//     Enc/Inputs/In/nDataIn1[0] <-> ENC Status compact/Counter value
//     Enc/Inputs/In/nDataIn2[0] <-> ENC Status compact/Latch value
//     Enc/Inputs/In/nState1 @bit 4 <-> ENC Status compact/Status/Counter overflow
//     Enc/Inputs/In/nState1 @bit 3 <-> ENC Status compact/Status/Counter underflow
//     Enc/Inputs/In/nState1 @bit 7 <-> ENC Status compact/Status/Extrapolation stall
//     Enc/Inputs/In/nState1 <-> ENC Status compact/Status/Latch C valid
//     Enc/Inputs/In/nState1 @bit 1 <-> ENC Status compact/Status/Latch extern valid
//     Enc/Inputs/In/nState1 @bit 2 <-> ENC Status compact/Status/Set counter done
//     Enc/Inputs/In/nState2 @bit 4 <-> ENC Status compact/Status/Status of extern latch
//     Enc/Inputs/In/nState2 <-> ENC Status compact/Status/Status of input A
//     Enc/Inputs/In/nState2 @bit 1 <-> ENC Status compact/Status/Status of input B
//     Enc/Inputs/In/nState2 @bit 2 <-> ENC Status compact/Status/Status of input C
//     Enc/Inputs/In/nState2 @bit 5 <-> ENC Status compact/Status/Sync error
//     Enc/Inputs/In/nState2 @bit 7 <-> ENC Status compact/Status/TxPDO Toggle
//     Enc/Inputs/In/nState4 @bit 1 <-> WcState/InputToggle
//     Enc/Inputs/In/nState4 <-> WcState/WcState
//     Enc/Outputs/Out/nCtrl1 <-> ENC Control compact/Control/Enable latch C
//     Enc/Outputs/Out/nCtrl1 @bit 3 <-> ENC Control compact/Control/Enable latch extern on negative edge
//     Enc/Outputs/Out/nCtrl1 @bit 1 <-> ENC Control compact/Control/Enable latch extern on positive edge
//     Enc/Outputs/Out/nCtrl1 @bit 2 <-> ENC Control compact/Control/Set counter
//     Enc/Outputs/Out/nDataOut1[0] <-> ENC Control compact/Set counter value
//   (this object) <-> Device 1 (EtherCAT)/Term 5 (EK1200)/Term 6 (EK1122-0080)/DRL02-EK0 (EK1101-0080)/DRL02-E21 (EL7041)
//     Drive/Inputs/In/nState1 @bit 3 <-> STM Status/Status/Error
//     Drive/Inputs/In/nState1 @bit 5 <-> STM Status/Status/Moving negative
//     Drive/Inputs/In/nState1 @bit 4 <-> STM Status/Status/Moving positive
//     Drive/Inputs/In/nState1 @bit 1 <-> STM Status/Status/Ready
//     Drive/Inputs/In/nState1 <-> STM Status/Status/Ready to enable
//     Drive/Inputs/In/nState1 @bit 6 <-> STM Status/Status/Torque reduced
//     Drive/Inputs/In/nState1 @bit 2 <-> STM Status/Status/Warning
//     Drive/Inputs/In/nState2 @bit 3 <-> STM Status/Status/Digital input 1
//     Drive/Inputs/In/nState2 @bit 4 <-> STM Status/Status/Digital input 2
//     Drive/Inputs/In/nState2 @bit 5 <-> STM Status/Status/Sync error
//     Drive/Inputs/In/nState2 @bit 7 <-> STM Status/Status/TxPDO Toggle
//     Drive/Inputs/In/nState4 @bit 1 <-> WcState/InputToggle
//     Drive/Inputs/In/nState4 <-> WcState/WcState
//     Drive/Outputs/Out/nCtrl1 <-> STM Control/Control/Enable
//     Drive/Outputs/Out/nCtrl1 @bit 2 <-> STM Control/Control/Reduce torque
//     Drive/Outputs/Out/nCtrl1 @bit 1 <-> STM Control/Control/Reset
//     Drive/Outputs/Out/nDataOut2[0] <-> STM Velocity/Velocity
//     Enc/Inputs/In/nDataIn1[0] <-> ENC Status compact/Counter value
//     Enc/Inputs/In/nDataIn2[0] <-> ENC Status compact/Latch value
//     Enc/Inputs/In/nState1 @bit 4 <-> ENC Status compact/Status/Counter overflow
//     Enc/Inputs/In/nState1 @bit 3 <-> ENC Status compact/Status/Counter underflow
//     Enc/Inputs/In/nState1 @bit 7 <-> ENC Status compact/Status/Extrapolation stall
//     Enc/Inputs/In/nState1 <-> ENC Status compact/Status/Latch C valid
//     Enc/Inputs/In/nState1 @bit 1 <-> ENC Status compact/Status/Latch extern valid
//     Enc/Inputs/In/nState1 @bit 2 <-> ENC Status compact/Status/Set counter done
//     Enc/Inputs/In/nState2 @bit 4 <-> ENC Status compact/Status/Status of extern latch
//     Enc/Inputs/In/nState2 <-> ENC Status compact/Status/Status of input A
//     Enc/Inputs/In/nState2 @bit 1 <-> ENC Status compact/Status/Status of input B
//     Enc/Inputs/In/nState2 @bit 2 <-> ENC Status compact/Status/Status of input C
//     Enc/Inputs/In/nState2 @bit 5 <-> ENC Status compact/Status/Sync error
//     Enc/Inputs/In/nState2 @bit 7 <-> ENC Status compact/Status/TxPDO Toggle
//     Enc/Inputs/In/nState4 @bit 1 <-> WcState/InputToggle
//     Enc/Inputs/In/nState4 <-> WcState/WcState
//     Enc/Outputs/Out/nCtrl1 <-> ENC Control compact/Control/Enable latch C
//     Enc/Outputs/Out/nCtrl1 @bit 3 <-> ENC Control compact/Control/Enable latch extern on negative edge
//     Enc/Outputs/Out/nCtrl1 @bit 1 <-> ENC Control compact/Control/Enable latch extern on positive edge
//     Enc/Outputs/Out/nCtrl1 @bit 2 <-> ENC Control compact/Control/Set counter
//     Enc/Outputs/Out/nDataOut1[0] <-> ENC Control compact/Set counter value
//   (this object) <-> Device 1 (EtherCAT)/Term 5 (EK1200)/Term 6 (EK1122-0080)/DRL02-EK0 (EK1101-0080)/DRL02-E1 (EL7031)
//     Drive/Inputs/In/nState1 @bit 3 <-> STM Status/Status/Error
//     Drive/Inputs/In/nState1 @bit 5 <-> STM Status/Status/Moving negative
//     Drive/Inputs/In/nState1 @bit 4 <-> STM Status/Status/Moving positive
//     Drive/Inputs/In/nState1 @bit 1 <-> STM Status/Status/Ready
//     Drive/Inputs/In/nState1 <-> STM Status/Status/Ready to enable
//     Drive/Inputs/In/nState1 @bit 6 <-> STM Status/Status/Torque reduced
//     Drive/Inputs/In/nState1 @bit 2 <-> STM Status/Status/Warning
//     Drive/Inputs/In/nState2 @bit 3 <-> STM Status/Status/Digital input 1
//     Drive/Inputs/In/nState2 @bit 4 <-> STM Status/Status/Digital input 2
//     Drive/Inputs/In/nState2 @bit 5 <-> STM Status/Status/Sync error
//     Drive/Inputs/In/nState2 @bit 7 <-> STM Status/Status/TxPDO Toggle
//     Drive/Inputs/In/nState4 @bit 1 <-> WcState/InputToggle
//     Drive/Inputs/In/nState4 <-> WcState/WcState
//     Drive/Outputs/Out/nCtrl1 <-> STM Control/Control/Enable
//     Drive/Outputs/Out/nCtrl1 @bit 2 <-> STM Control/Control/Reduce torque
//     Drive/Outputs/Out/nCtrl1 @bit 1 <-> STM Control/Control/Reset
//     Drive/Outputs/Out/nDataOut2[0] <-> STM Velocity/Velocity
//   (this object) <-> Device 1 (EtherCAT)/Term 5 (EK1200)/Term 6 (EK1122-0080)/DRL02-EK0 (EK1101-0080)/DRL02-E2 (EL5042)
//     Enc/Inputs/In/nComState @bit 1 <-> WcState/InputToggle
//     Enc/Inputs/In/nComState <-> WcState/WcState
//     Enc/Inputs/In/nDataIn1 <-> FB Inputs Channel 1/Position
//     Enc/Inputs/In/nDataIn1 <-> FB Inputs Channel 2/Position
//     Enc/Inputs/In/nState1 @bit 12 <-> FB Inputs Channel 1/Status/Diag
//     Enc/Inputs/In/nState1 @bit 12 <-> FB Inputs Channel 2/Status/Diag
//     Enc/Inputs/In/nState1 @bit 1 <-> FB Inputs Channel 1/Status/Error
//     Enc/Inputs/In/nState1 @bit 1 <-> FB Inputs Channel 2/Status/Error
//     Enc/Inputs/In/nState1 @bit 14 <-> FB Inputs Channel 1/Status/Input cycle counter
//     Enc/Inputs/In/nState1 @bit 14 <-> FB Inputs Channel 2/Status/Input cycle counter
//     Enc/Inputs/In/nState1 @bit 2 <-> FB Inputs Channel 1/Status/Ready
//     Enc/Inputs/In/nState1 @bit 2 <-> FB Inputs Channel 2/Status/Ready
//     Enc/Inputs/In/nState1 @bit 13 <-> FB Inputs Channel 1/Status/TxPDO State
//     Enc/Inputs/In/nState1 @bit 13 <-> FB Inputs Channel 2/Status/TxPDO State
//     Enc/Inputs/In/nState1 <-> FB Inputs Channel 1/Status/Warning
//     Enc/Inputs/In/nState1 <-> FB Inputs Channel 2/Status/Warning
//   (this object) <-> Device 1 (EtherCAT)/Term 5 (EK1200)/Term 6 (EK1122-0080)/DRL02-EK0 (EK1101-0080)/DRL02-E3 (EL7031)
//     Drive/Inputs/In/nState1 @bit 3 <-> STM Status/Status/Error
//     Drive/Inputs/In/nState1 @bit 5 <-> STM Status/Status/Moving negative
//     Drive/Inputs/In/nState1 @bit 4 <-> STM Status/Status/Moving positive
//     Drive/Inputs/In/nState1 @bit 1 <-> STM Status/Status/Ready
//     Drive/Inputs/In/nState1 <-> STM Status/Status/Ready to enable
//     Drive/Inputs/In/nState1 @bit 6 <-> STM Status/Status/Torque reduced
//     Drive/Inputs/In/nState1 @bit 2 <-> STM Status/Status/Warning
//     Drive/Inputs/In/nState2 @bit 3 <-> STM Status/Status/Digital input 1
//     Drive/Inputs/In/nState2 @bit 4 <-> STM Status/Status/Digital input 2
//     Drive/Inputs/In/nState2 @bit 5 <-> STM Status/Status/Sync error
//     Drive/Inputs/In/nState2 @bit 7 <-> STM Status/Status/TxPDO Toggle
//     Drive/Inputs/In/nState4 @bit 1 <-> WcState/InputToggle
//     Drive/Inputs/In/nState4 <-> WcState/WcState
//     Drive/Outputs/Out/nCtrl1 <-> STM Control/Control/Enable
//     Drive/Outputs/Out/nCtrl1 @bit 2 <-> STM Control/Control/Reduce torque
//     Drive/Outputs/Out/nCtrl1 @bit 1 <-> STM Control/Control/Reset
//     Drive/Outputs/Out/nDataOut2[0] <-> STM Velocity/Velocity
//   (this object) <-> Device 1 (EtherCAT)/Term 5 (EK1200)/Term 6 (EK1122-0080)/DRL02-EK0 (EK1101-0080)/DRL02-E4 (EL7031)
//     Drive/Inputs/In/nState1 @bit 3 <-> STM Status/Status/Error
//     Drive/Inputs/In/nState1 @bit 5 <-> STM Status/Status/Moving negative
//     Drive/Inputs/In/nState1 @bit 4 <-> STM Status/Status/Moving positive
//     Drive/Inputs/In/nState1 @bit 1 <-> STM Status/Status/Ready
//     Drive/Inputs/In/nState1 <-> STM Status/Status/Ready to enable
//     Drive/Inputs/In/nState1 @bit 6 <-> STM Status/Status/Torque reduced
//     Drive/Inputs/In/nState1 @bit 2 <-> STM Status/Status/Warning
//     Drive/Inputs/In/nState2 @bit 3 <-> STM Status/Status/Digital input 1
//     Drive/Inputs/In/nState2 @bit 4 <-> STM Status/Status/Digital input 2
//     Drive/Inputs/In/nState2 @bit 5 <-> STM Status/Status/Sync error
//     Drive/Inputs/In/nState2 @bit 7 <-> STM Status/Status/TxPDO Toggle
//     Drive/Inputs/In/nState4 @bit 1 <-> WcState/InputToggle
//     Drive/Inputs/In/nState4 <-> WcState/WcState
//     Drive/Outputs/Out/nCtrl1 <-> STM Control/Control/Enable
//     Drive/Outputs/Out/nCtrl1 @bit 2 <-> STM Control/Control/Reduce torque
//     Drive/Outputs/Out/nCtrl1 @bit 1 <-> STM Control/Control/Reset
//     Drive/Outputs/Out/nDataOut2[0] <-> STM Velocity/Velocity
//   (this object) <-> Device 1 (EtherCAT)/Term 5 (EK1200)/Term 6 (EK1122-0080)/DRL02-EK0 (EK1101-0080)/DRL02-E5 (EL5042)
//     Enc/Inputs/In/nComState @bit 1 <-> WcState/InputToggle
//     Enc/Inputs/In/nComState <-> WcState/WcState
//     Enc/Inputs/In/nDataIn1 <-> FB Inputs Channel 1/Position
//     Enc/Inputs/In/nDataIn1 <-> FB Inputs Channel 2/Position
//     Enc/Inputs/In/nState1 @bit 12 <-> FB Inputs Channel 1/Status/Diag
//     Enc/Inputs/In/nState1 @bit 12 <-> FB Inputs Channel 2/Status/Diag
//     Enc/Inputs/In/nState1 @bit 1 <-> FB Inputs Channel 1/Status/Error
//     Enc/Inputs/In/nState1 @bit 1 <-> FB Inputs Channel 2/Status/Error
//     Enc/Inputs/In/nState1 @bit 14 <-> FB Inputs Channel 1/Status/Input cycle counter
//     Enc/Inputs/In/nState1 @bit 14 <-> FB Inputs Channel 2/Status/Input cycle counter
//     Enc/Inputs/In/nState1 @bit 2 <-> FB Inputs Channel 1/Status/Ready
//     Enc/Inputs/In/nState1 @bit 2 <-> FB Inputs Channel 2/Status/Ready
//     Enc/Inputs/In/nState1 @bit 13 <-> FB Inputs Channel 1/Status/TxPDO State
//     Enc/Inputs/In/nState1 @bit 13 <-> FB Inputs Channel 2/Status/TxPDO State
//     Enc/Inputs/In/nState1 <-> FB Inputs Channel 1/Status/Warning
//     Enc/Inputs/In/nState1 <-> FB Inputs Channel 2/Status/Warning
//   (this object) <-> Device 1 (EtherCAT)/Term 5 (EK1200)/Term 6 (EK1122-0080)/DRL02-EK0 (EK1101-0080)/DRL02-E6 (EL7031)
//     Drive/Inputs/In/nState1 @bit 3 <-> STM Status/Status/Error
//     Drive/Inputs/In/nState1 @bit 5 <-> STM Status/Status/Moving negative
//     Drive/Inputs/In/nState1 @bit 4 <-> STM Status/Status/Moving positive
//     Drive/Inputs/In/nState1 @bit 1 <-> STM Status/Status/Ready
//     Drive/Inputs/In/nState1 <-> STM Status/Status/Ready to enable
//     Drive/Inputs/In/nState1 @bit 6 <-> STM Status/Status/Torque reduced
//     Drive/Inputs/In/nState1 @bit 2 <-> STM Status/Status/Warning
//     Drive/Inputs/In/nState2 @bit 3 <-> STM Status/Status/Digital input 1
//     Drive/Inputs/In/nState2 @bit 4 <-> STM Status/Status/Digital input 2
//     Drive/Inputs/In/nState2 @bit 5 <-> STM Status/Status/Sync error
//     Drive/Inputs/In/nState2 @bit 7 <-> STM Status/Status/TxPDO Toggle
//     Drive/Inputs/In/nState4 @bit 1 <-> WcState/InputToggle
//     Drive/Inputs/In/nState4 <-> WcState/WcState
//     Drive/Outputs/Out/nCtrl1 <-> STM Control/Control/Enable
//     Drive/Outputs/Out/nCtrl1 @bit 2 <-> STM Control/Control/Reduce torque
//     Drive/Outputs/Out/nCtrl1 @bit 1 <-> STM Control/Control/Reset
//     Drive/Outputs/Out/nDataOut2[0] <-> STM Velocity/Velocity
//   (this object) <-> Device 1 (EtherCAT)/Term 5 (EK1200)/Term 6 (EK1122-0080)/DRL02-EK0 (EK1101-0080)/DRL02-E7 (EL7031)
//     Drive/Inputs/In/nState1 @bit 3 <-> STM Status/Status/Error
//     Drive/Inputs/In/nState1 @bit 5 <-> STM Status/Status/Moving negative
//     Drive/Inputs/In/nState1 @bit 4 <-> STM Status/Status/Moving positive
//     Drive/Inputs/In/nState1 @bit 1 <-> STM Status/Status/Ready
//     Drive/Inputs/In/nState1 <-> STM Status/Status/Ready to enable
//     Drive/Inputs/In/nState1 @bit 6 <-> STM Status/Status/Torque reduced
//     Drive/Inputs/In/nState1 @bit 2 <-> STM Status/Status/Warning
//     Drive/Inputs/In/nState2 @bit 3 <-> STM Status/Status/Digital input 1
//     Drive/Inputs/In/nState2 @bit 4 <-> STM Status/Status/Digital input 2
//     Drive/Inputs/In/nState2 @bit 5 <-> STM Status/Status/Sync error
//     Drive/Inputs/In/nState2 @bit 7 <-> STM Status/Status/TxPDO Toggle
//     Drive/Inputs/In/nState4 @bit 1 <-> WcState/InputToggle
//     Drive/Inputs/In/nState4 <-> WcState/WcState
//     Drive/Outputs/Out/nCtrl1 <-> STM Control/Control/Enable
//     Drive/Outputs/Out/nCtrl1 @bit 2 <-> STM Control/Control/Reduce torque
//     Drive/Outputs/Out/nCtrl1 @bit 1 <-> STM Control/Control/Reset
//     Drive/Outputs/Out/nDataOut2[0] <-> STM Velocity/Velocity
//   (this object) <-> Device 1 (EtherCAT)/Term 5 (EK1200)/Term 6 (EK1122-0080)/DRL02-EK0 (EK1101-0080)/DRL02-E8 (EL5042)
//     Enc/Inputs/In/nComState @bit 1 <-> WcState/InputToggle
//     Enc/Inputs/In/nComState <-> WcState/WcState
//     Enc/Inputs/In/nDataIn1 <-> FB Inputs Channel 1/Position
//     Enc/Inputs/In/nDataIn1 <-> FB Inputs Channel 2/Position
//     Enc/Inputs/In/nState1 @bit 12 <-> FB Inputs Channel 1/Status/Diag
//     Enc/Inputs/In/nState1 @bit 12 <-> FB Inputs Channel 2/Status/Diag
//     Enc/Inputs/In/nState1 @bit 1 <-> FB Inputs Channel 1/Status/Error
//     Enc/Inputs/In/nState1 @bit 1 <-> FB Inputs Channel 2/Status/Error
//     Enc/Inputs/In/nState1 @bit 14 <-> FB Inputs Channel 1/Status/Input cycle counter
//     Enc/Inputs/In/nState1 @bit 14 <-> FB Inputs Channel 2/Status/Input cycle counter
//     Enc/Inputs/In/nState1 @bit 2 <-> FB Inputs Channel 1/Status/Ready
//     Enc/Inputs/In/nState1 @bit 2 <-> FB Inputs Channel 2/Status/Ready
//     Enc/Inputs/In/nState1 @bit 13 <-> FB Inputs Channel 1/Status/TxPDO State
//     Enc/Inputs/In/nState1 @bit 13 <-> FB Inputs Channel 2/Status/TxPDO State
//     Enc/Inputs/In/nState1 <-> FB Inputs Channel 1/Status/Warning
//     Enc/Inputs/In/nState1 <-> FB Inputs Channel 2/Status/Warning
//   (this object) <-> Device 1 (EtherCAT)/Term 5 (EK1200)/Term 6 (EK1122-0080)/DRL02-EK0 (EK1101-0080)/DRL02-E9 (EL7031)
//     Drive/Inputs/In/nState1 @bit 3 <-> STM Status/Status/Error
//     Drive/Inputs/In/nState1 @bit 5 <-> STM Status/Status/Moving negative
//     Drive/Inputs/In/nState1 @bit 4 <-> STM Status/Status/Moving positive
//     Drive/Inputs/In/nState1 @bit 1 <-> STM Status/Status/Ready
//     Drive/Inputs/In/nState1 <-> STM Status/Status/Ready to enable
//     Drive/Inputs/In/nState1 @bit 6 <-> STM Status/Status/Torque reduced
//     Drive/Inputs/In/nState1 @bit 2 <-> STM Status/Status/Warning
//     Drive/Inputs/In/nState2 @bit 3 <-> STM Status/Status/Digital input 1
//     Drive/Inputs/In/nState2 @bit 4 <-> STM Status/Status/Digital input 2
//     Drive/Inputs/In/nState2 @bit 5 <-> STM Status/Status/Sync error
//     Drive/Inputs/In/nState2 @bit 7 <-> STM Status/Status/TxPDO Toggle
//     Drive/Inputs/In/nState4 @bit 1 <-> WcState/InputToggle
//     Drive/Inputs/In/nState4 <-> WcState/WcState
//     Drive/Outputs/Out/nCtrl1 <-> STM Control/Control/Enable
//     Drive/Outputs/Out/nCtrl1 @bit 2 <-> STM Control/Control/Reduce torque
//     Drive/Outputs/Out/nCtrl1 @bit 1 <-> STM Control/Control/Reset
//     Drive/Outputs/Out/nDataOut2[0] <-> STM Velocity/Velocity
//   (this object) <-> Device 1 (EtherCAT)/Term 5 (EK1200)/Term 6 (EK1122-0080)/DRL02-EK0 (EK1101-0080)/DRL02-E11 (EL7031)
//     Drive/Inputs/In/nState1 @bit 3 <-> STM Status/Status/Error
//     Drive/Inputs/In/nState1 @bit 5 <-> STM Status/Status/Moving negative
//     Drive/Inputs/In/nState1 @bit 4 <-> STM Status/Status/Moving positive
//     Drive/Inputs/In/nState1 @bit 1 <-> STM Status/Status/Ready
//     Drive/Inputs/In/nState1 <-> STM Status/Status/Ready to enable
//     Drive/Inputs/In/nState1 @bit 6 <-> STM Status/Status/Torque reduced
//     Drive/Inputs/In/nState1 @bit 2 <-> STM Status/Status/Warning
//     Drive/Inputs/In/nState2 @bit 3 <-> STM Status/Status/Digital input 1
//     Drive/Inputs/In/nState2 @bit 4 <-> STM Status/Status/Digital input 2
//     Drive/Inputs/In/nState2 @bit 5 <-> STM Status/Status/Sync error
//     Drive/Inputs/In/nState2 @bit 7 <-> STM Status/Status/TxPDO Toggle
//     Drive/Inputs/In/nState4 @bit 1 <-> WcState/InputToggle
//     Drive/Inputs/In/nState4 <-> WcState/WcState
//     Drive/Outputs/Out/nCtrl1 <-> STM Control/Control/Enable
//     Drive/Outputs/Out/nCtrl1 @bit 2 <-> STM Control/Control/Reduce torque
//     Drive/Outputs/Out/nCtrl1 @bit 1 <-> STM Control/Control/Reset
//     Drive/Outputs/Out/nDataOut2[0] <-> STM Velocity/Velocity
//   (this object) <-> Device 1 (EtherCAT)/Term 5 (EK1200)/Term 6 (EK1122-0080)/DRL02-EK0 (EK1101-0080)/DRL02-E12 (EL5042)
//     Enc/Inputs/In/nComState @bit 1 <-> WcState/InputToggle
//     Enc/Inputs/In/nComState <-> WcState/WcState
//     Enc/Inputs/In/nDataIn1 <-> FB Inputs Channel 1/Position
//     Enc/Inputs/In/nDataIn1 <-> FB Inputs Channel 2/Position
//     Enc/Inputs/In/nState1 @bit 12 <-> FB Inputs Channel 1/Status/Diag
//     Enc/Inputs/In/nState1 @bit 12 <-> FB Inputs Channel 2/Status/Diag
//     Enc/Inputs/In/nState1 @bit 1 <-> FB Inputs Channel 1/Status/Error
//     Enc/Inputs/In/nState1 @bit 1 <-> FB Inputs Channel 2/Status/Error
//     Enc/Inputs/In/nState1 @bit 14 <-> FB Inputs Channel 1/Status/Input cycle counter
//     Enc/Inputs/In/nState1 @bit 14 <-> FB Inputs Channel 2/Status/Input cycle counter
//     Enc/Inputs/In/nState1 @bit 2 <-> FB Inputs Channel 1/Status/Ready
//     Enc/Inputs/In/nState1 @bit 2 <-> FB Inputs Channel 2/Status/Ready
//     Enc/Inputs/In/nState1 @bit 13 <-> FB Inputs Channel 1/Status/TxPDO State
//     Enc/Inputs/In/nState1 @bit 13 <-> FB Inputs Channel 2/Status/TxPDO State
//     Enc/Inputs/In/nState1 <-> FB Inputs Channel 1/Status/Warning
//     Enc/Inputs/In/nState1 <-> FB Inputs Channel 2/Status/Warning
//   (this object) <-> Device 1 (EtherCAT)/Term 5 (EK1200)/Term 6 (EK1122-0080)/DRL02-EK0 (EK1101-0080)/DRL02-E13 (EL7041)
//     Drive/Inputs/In/nState1 @bit 3 <-> STM Status/Status/Error
//     Drive/Inputs/In/nState1 @bit 5 <-> STM Status/Status/Moving negative
//     Drive/Inputs/In/nState1 @bit 4 <-> STM Status/Status/Moving positive
//     Drive/Inputs/In/nState1 @bit 1 <-> STM Status/Status/Ready
//     Drive/Inputs/In/nState1 <-> STM Status/Status/Ready to enable
//     Drive/Inputs/In/nState1 @bit 6 <-> STM Status/Status/Torque reduced
//     Drive/Inputs/In/nState1 @bit 2 <-> STM Status/Status/Warning
//     Drive/Inputs/In/nState2 @bit 3 <-> STM Status/Status/Digital input 1
//     Drive/Inputs/In/nState2 @bit 4 <-> STM Status/Status/Digital input 2
//     Drive/Inputs/In/nState2 @bit 5 <-> STM Status/Status/Sync error
//     Drive/Inputs/In/nState2 @bit 7 <-> STM Status/Status/TxPDO Toggle
//     Drive/Inputs/In/nState4 @bit 1 <-> WcState/InputToggle
//     Drive/Inputs/In/nState4 <-> WcState/WcState
//     Drive/Outputs/Out/nCtrl1 <-> STM Control/Control/Enable
//     Drive/Outputs/Out/nCtrl1 @bit 2 <-> STM Control/Control/Reduce torque
//     Drive/Outputs/Out/nCtrl1 @bit 1 <-> STM Control/Control/Reset
//     Drive/Outputs/Out/nDataOut2[0] <-> STM Velocity/Velocity
//   (this object) <-> Device 1 (EtherCAT)/Term 5 (EK1200)/Term 6 (EK1122-0080)/DRL02-EK0 (EK1101-0080)/Term 63 (EL7031)
//     Drive/Inputs/In/nState1 @bit 3 <-> STM Status/Status/Error
//     Drive/Inputs/In/nState1 @bit 5 <-> STM Status/Status/Moving negative
//     Drive/Inputs/In/nState1 @bit 4 <-> STM Status/Status/Moving positive
//     Drive/Inputs/In/nState1 @bit 1 <-> STM Status/Status/Ready
//     Drive/Inputs/In/nState1 <-> STM Status/Status/Ready to enable
//     Drive/Inputs/In/nState1 @bit 6 <-> STM Status/Status/Torque reduced
//     Drive/Inputs/In/nState1 @bit 2 <-> STM Status/Status/Warning
//     Drive/Inputs/In/nState2 @bit 3 <-> STM Status/Status/Digital input 1
//     Drive/Inputs/In/nState2 @bit 4 <-> STM Status/Status/Digital input 2
//     Drive/Inputs/In/nState2 @bit 5 <-> STM Status/Status/Sync error
//     Drive/Inputs/In/nState2 @bit 7 <-> STM Status/Status/TxPDO Toggle
//     Drive/Inputs/In/nState4 @bit 1 <-> WcState/InputToggle
//     Drive/Inputs/In/nState4 <-> WcState/WcState
//     Drive/Outputs/Out/nCtrl1 <-> STM Control/Control/Enable
//     Drive/Outputs/Out/nCtrl1 @bit 2 <-> STM Control/Control/Reduce torque
//     Drive/Outputs/Out/nCtrl1 @bit 1 <-> STM Control/Control/Reset
//     Drive/Outputs/Out/nDataOut2[0] <-> STM Velocity/Velocity
//     Enc/Inputs/In/nDataIn1[0] <-> ENC Status compact/Counter value
//     Enc/Inputs/In/nDataIn2[0] <-> ENC Status compact/Latch value
//     Enc/Inputs/In/nState1 @bit 4 <-> ENC Status compact/Status/Counter overflow
//     Enc/Inputs/In/nState1 @bit 3 <-> ENC Status compact/Status/Counter underflow
//     Enc/Inputs/In/nState1 @bit 1 <-> ENC Status compact/Status/Latch extern valid
//     Enc/Inputs/In/nState1 @bit 2 <-> ENC Status compact/Status/Set counter done
//     Enc/Inputs/In/nState2 @bit 4 <-> ENC Status compact/Status/Status of extern latch
//     Enc/Inputs/In/nState2 @bit 5 <-> ENC Status compact/Status/Sync error
//     Enc/Inputs/In/nState2 @bit 7 <-> ENC Status compact/Status/TxPDO Toggle
//     Enc/Inputs/In/nState4 @bit 1 <-> WcState/InputToggle
//     Enc/Inputs/In/nState4 <-> WcState/WcState
//     Enc/Outputs/Out/nCtrl1 @bit 3 <-> ENC Control compact/Control/Enable latch extern on negative edge
//     Enc/Outputs/Out/nCtrl1 @bit 1 <-> ENC Control compact/Control/Enable latch extern on positive edge
//     Enc/Outputs/Out/nCtrl1 @bit 2 <-> ENC Control compact/Control/Set counter
//     Enc/Outputs/Out/nDataOut1[0] <-> ENC Control compact/Set counter value
//   (this object) <-> Device 1 (EtherCAT)/Term 5 (EK1200)/Term 6 (EK1122-0080)/DRL02-EK0 (EK1101-0080)/Term 66 (EL7031)
//     Drive/Inputs/In/nState1 @bit 3 <-> STM Status/Status/Error
//     Drive/Inputs/In/nState1 @bit 5 <-> STM Status/Status/Moving negative
//     Drive/Inputs/In/nState1 @bit 4 <-> STM Status/Status/Moving positive
//     Drive/Inputs/In/nState1 @bit 1 <-> STM Status/Status/Ready
//     Drive/Inputs/In/nState1 <-> STM Status/Status/Ready to enable
//     Drive/Inputs/In/nState1 @bit 6 <-> STM Status/Status/Torque reduced
//     Drive/Inputs/In/nState1 @bit 2 <-> STM Status/Status/Warning
//     Drive/Inputs/In/nState2 @bit 3 <-> STM Status/Status/Digital input 1
//     Drive/Inputs/In/nState2 @bit 4 <-> STM Status/Status/Digital input 2
//     Drive/Inputs/In/nState2 @bit 5 <-> STM Status/Status/Sync error
//     Drive/Inputs/In/nState2 @bit 7 <-> STM Status/Status/TxPDO Toggle
//     Drive/Inputs/In/nState4 @bit 1 <-> WcState/InputToggle
//     Drive/Inputs/In/nState4 <-> WcState/WcState
//     Drive/Outputs/Out/nCtrl1 <-> STM Control/Control/Enable
//     Drive/Outputs/Out/nCtrl1 @bit 2 <-> STM Control/Control/Reduce torque
//     Drive/Outputs/Out/nCtrl1 @bit 1 <-> STM Control/Control/Reset
//     Drive/Outputs/Out/nDataOut2[0] <-> STM Velocity/Velocity
//     Enc/Inputs/In/nDataIn1[0] <-> ENC Status compact/Counter value
//     Enc/Inputs/In/nDataIn2[0] <-> ENC Status compact/Latch value
//     Enc/Inputs/In/nState1 @bit 4 <-> ENC Status compact/Status/Counter overflow
//     Enc/Inputs/In/nState1 @bit 3 <-> ENC Status compact/Status/Counter underflow
//     Enc/Inputs/In/nState1 @bit 1 <-> ENC Status compact/Status/Latch extern valid
//     Enc/Inputs/In/nState1 @bit 2 <-> ENC Status compact/Status/Set counter done
//     Enc/Inputs/In/nState2 @bit 4 <-> ENC Status compact/Status/Status of extern latch
//     Enc/Inputs/In/nState2 @bit 5 <-> ENC Status compact/Status/Sync error
//     Enc/Inputs/In/nState2 @bit 7 <-> ENC Status compact/Status/TxPDO Toggle
//     Enc/Inputs/In/nState4 @bit 1 <-> WcState/InputToggle
//     Enc/Inputs/In/nState4 <-> WcState/WcState
//     Enc/Outputs/Out/nCtrl1 @bit 3 <-> ENC Control compact/Control/Enable latch extern on negative edge
//     Enc/Outputs/Out/nCtrl1 @bit 1 <-> ENC Control compact/Control/Enable latch extern on positive edge
//     Enc/Outputs/Out/nCtrl1 @bit 2 <-> ENC Control compact/Control/Set counter
//     Enc/Outputs/Out/nDataOut1[0] <-> ENC Control compact/Set counter value
//   (this object) <-> Device 1 (EtherCAT)/Term 5 (EK1200)/Term 6 (EK1122-0080)/DRL02-EK0 (EK1101-0080)/Term 67 (EL7031)
//     Drive/Inputs/In/nState1 @bit 3 <-> STM Status/Status/Error
//     Drive/Inputs/In/nState1 @bit 5 <-> STM Status/Status/Moving negative
//     Drive/Inputs/In/nState1 @bit 4 <-> STM Status/Status/Moving positive
//     Drive/Inputs/In/nState1 @bit 1 <-> STM Status/Status/Ready
//     Drive/Inputs/In/nState1 <-> STM Status/Status/Ready to enable
//     Drive/Inputs/In/nState1 @bit 6 <-> STM Status/Status/Torque reduced
//     Drive/Inputs/In/nState1 @bit 2 <-> STM Status/Status/Warning
//     Drive/Inputs/In/nState2 @bit 3 <-> STM Status/Status/Digital input 1
//     Drive/Inputs/In/nState2 @bit 4 <-> STM Status/Status/Digital input 2
//     Drive/Inputs/In/nState2 @bit 5 <-> STM Status/Status/Sync error
//     Drive/Inputs/In/nState2 @bit 7 <-> STM Status/Status/TxPDO Toggle
//     Drive/Inputs/In/nState4 @bit 1 <-> WcState/InputToggle
//     Drive/Inputs/In/nState4 <-> WcState/WcState
//     Drive/Outputs/Out/nCtrl1 <-> STM Control/Control/Enable
//     Drive/Outputs/Out/nCtrl1 @bit 2 <-> STM Control/Control/Reduce torque
//     Drive/Outputs/Out/nCtrl1 @bit 1 <-> STM Control/Control/Reset
//     Drive/Outputs/Out/nDataOut2[0] <-> STM Velocity/Velocity
//     Enc/Inputs/In/nDataIn1[0] <-> ENC Status compact/Counter value
//     Enc/Inputs/In/nDataIn2[0] <-> ENC Status compact/Latch value
//     Enc/Inputs/In/nState1 @bit 4 <-> ENC Status compact/Status/Counter overflow
//     Enc/Inputs/In/nState1 @bit 3 <-> ENC Status compact/Status/Counter underflow
//     Enc/Inputs/In/nState1 @bit 1 <-> ENC Status compact/Status/Latch extern valid
//     Enc/Inputs/In/nState1 @bit 2 <-> ENC Status compact/Status/Set counter done
//     Enc/Inputs/In/nState2 @bit 4 <-> ENC Status compact/Status/Status of extern latch
//     Enc/Inputs/In/nState2 @bit 5 <-> ENC Status compact/Status/Sync error
//     Enc/Inputs/In/nState2 @bit 7 <-> ENC Status compact/Status/TxPDO Toggle
//     Enc/Inputs/In/nState4 @bit 1 <-> WcState/InputToggle
//     Enc/Inputs/In/nState4 <-> WcState/WcState
//     Enc/Outputs/Out/nCtrl1 @bit 3 <-> ENC Control compact/Control/Enable latch extern on negative edge
//     Enc/Outputs/Out/nCtrl1 @bit 1 <-> ENC Control compact/Control/Enable latch extern on positive edge
//     Enc/Outputs/Out/nCtrl1 @bit 2 <-> ENC Control compact/Control/Set counter
//     Enc/Outputs/Out/nDataOut1[0] <-> ENC Control compact/Set counter value
//   (this object) <-> Device 1 (EtherCAT)/Term 5 (EK1200)/Term 6 (EK1122-0080)/DRL02-EK0 (EK1101-0080)/DRL02-E17 (EL7031)
//     Drive/Inputs/In/nState1 @bit 3 <-> STM Status/Status/Error
//     Drive/Inputs/In/nState1 @bit 5 <-> STM Status/Status/Moving negative
//     Drive/Inputs/In/nState1 @bit 4 <-> STM Status/Status/Moving positive
//     Drive/Inputs/In/nState1 @bit 1 <-> STM Status/Status/Ready
//     Drive/Inputs/In/nState1 <-> STM Status/Status/Ready to enable
//     Drive/Inputs/In/nState1 @bit 6 <-> STM Status/Status/Torque reduced
//     Drive/Inputs/In/nState1 @bit 2 <-> STM Status/Status/Warning
//     Drive/Inputs/In/nState2 @bit 3 <-> STM Status/Status/Digital input 1
//     Drive/Inputs/In/nState2 @bit 4 <-> STM Status/Status/Digital input 2
//     Drive/Inputs/In/nState2 @bit 5 <-> STM Status/Status/Sync error
//     Drive/Inputs/In/nState2 @bit 7 <-> STM Status/Status/TxPDO Toggle
//     Drive/Inputs/In/nState4 @bit 1 <-> WcState/InputToggle
//     Drive/Inputs/In/nState4 <-> WcState/WcState
//     Drive/Outputs/Out/nCtrl1 <-> STM Control/Control/Enable
//     Drive/Outputs/Out/nCtrl1 @bit 2 <-> STM Control/Control/Reduce torque
//     Drive/Outputs/Out/nCtrl1 @bit 1 <-> STM Control/Control/Reset
//     Drive/Outputs/Out/nDataOut2[0] <-> STM Velocity/Velocity
//   (this object) <-> Device 1 (EtherCAT)/Term 5 (EK1200)/Term 6 (EK1122-0080)/DRL02-EK0 (EK1101-0080)/DRL02-E18 (EL5042)
//     Enc/Inputs/In/nComState @bit 1 <-> WcState/InputToggle
//     Enc/Inputs/In/nComState <-> WcState/WcState
//     Enc/Inputs/In/nDataIn1 <-> FB Inputs Channel 1/Position
//     Enc/Inputs/In/nDataIn1 <-> FB Inputs Channel 2/Position
//     Enc/Inputs/In/nState1 @bit 12 <-> FB Inputs Channel 1/Status/Diag
//     Enc/Inputs/In/nState1 @bit 12 <-> FB Inputs Channel 2/Status/Diag
//     Enc/Inputs/In/nState1 @bit 1 <-> FB Inputs Channel 1/Status/Error
//     Enc/Inputs/In/nState1 @bit 1 <-> FB Inputs Channel 2/Status/Error
//     Enc/Inputs/In/nState1 @bit 14 <-> FB Inputs Channel 1/Status/Input cycle counter
//     Enc/Inputs/In/nState1 @bit 14 <-> FB Inputs Channel 2/Status/Input cycle counter
//     Enc/Inputs/In/nState1 @bit 2 <-> FB Inputs Channel 1/Status/Ready
//     Enc/Inputs/In/nState1 @bit 2 <-> FB Inputs Channel 2/Status/Ready
//     Enc/Inputs/In/nState1 @bit 13 <-> FB Inputs Channel 1/Status/TxPDO State
//     Enc/Inputs/In/nState1 @bit 13 <-> FB Inputs Channel 2/Status/TxPDO State
//     Enc/Inputs/In/nState1 <-> FB Inputs Channel 1/Status/Warning
//     Enc/Inputs/In/nState1 <-> FB Inputs Channel 2/Status/Warning
//   (this object) <-> Device 1 (EtherCAT)/Term 5 (EK1200)/Term 6 (EK1122-0080)/DRL02-EK0 (EK1101-0080)/DRL02-E19 (EL7031)
//     Drive/Inputs/In/nState1 @bit 3 <-> STM Status/Status/Error
//     Drive/Inputs/In/nState1 @bit 5 <-> STM Status/Status/Moving negative
//     Drive/Inputs/In/nState1 @bit 4 <-> STM Status/Status/Moving positive
//     Drive/Inputs/In/nState1 @bit 1 <-> STM Status/Status/Ready
//     Drive/Inputs/In/nState1 <-> STM Status/Status/Ready to enable
//     Drive/Inputs/In/nState1 @bit 6 <-> STM Status/Status/Torque reduced
//     Drive/Inputs/In/nState1 @bit 2 <-> STM Status/Status/Warning
//     Drive/Inputs/In/nState2 @bit 3 <-> STM Status/Status/Digital input 1
//     Drive/Inputs/In/nState2 @bit 4 <-> STM Status/Status/Digital input 2
//     Drive/Inputs/In/nState2 @bit 5 <-> STM Status/Status/Sync error
//     Drive/Inputs/In/nState2 @bit 7 <-> STM Status/Status/TxPDO Toggle
//     Drive/Inputs/In/nState4 @bit 1 <-> WcState/InputToggle
//     Drive/Inputs/In/nState4 <-> WcState/WcState
//     Drive/Outputs/Out/nCtrl1 <-> STM Control/Control/Enable
//     Drive/Outputs/Out/nCtrl1 @bit 2 <-> STM Control/Control/Reduce torque
//     Drive/Outputs/Out/nCtrl1 @bit 1 <-> STM Control/Control/Reset
//     Drive/Outputs/Out/nDataOut2[0] <-> STM Velocity/Velocity
//   (this object) <-> Device 1 (EtherCAT)/Term 5 (EK1200)/Term 6 (EK1122-0080)/DRL02-EK0 (EK1101-0080)/DRL02-E24 (EL7031)
//     Drive/Inputs/In/nState1 @bit 3 <-> STM Status/Status/Error
//     Drive/Inputs/In/nState1 @bit 5 <-> STM Status/Status/Moving negative
//     Drive/Inputs/In/nState1 @bit 4 <-> STM Status/Status/Moving positive
//     Drive/Inputs/In/nState1 @bit 1 <-> STM Status/Status/Ready
//     Drive/Inputs/In/nState1 <-> STM Status/Status/Ready to enable
//     Drive/Inputs/In/nState1 @bit 6 <-> STM Status/Status/Torque reduced
//     Drive/Inputs/In/nState1 @bit 2 <-> STM Status/Status/Warning
//     Drive/Inputs/In/nState2 @bit 3 <-> STM Status/Status/Digital input 1
//     Drive/Inputs/In/nState2 @bit 4 <-> STM Status/Status/Digital input 2
//     Drive/Inputs/In/nState2 @bit 5 <-> STM Status/Status/Sync error
//     Drive/Inputs/In/nState2 @bit 7 <-> STM Status/Status/TxPDO Toggle
//     Drive/Inputs/In/nState4 @bit 1 <-> WcState/InputToggle
//     Drive/Inputs/In/nState4 <-> WcState/WcState
//     Drive/Outputs/Out/nCtrl1 <-> STM Control/Control/Enable
//     Drive/Outputs/Out/nCtrl1 @bit 2 <-> STM Control/Control/Reduce torque
//     Drive/Outputs/Out/nCtrl1 @bit 1 <-> STM Control/Control/Reset
//     Drive/Outputs/Out/nDataOut2[0] <-> STM Velocity/Velocity
//   (this object) <-> Device 1 (EtherCAT)/Term 5 (EK1200)/Term 6 (EK1122-0080)/DRL02-EK0 (EK1101-0080)/Term 91 (EL5112)
//     Enc/Inputs/In/nDataIn1 <-> ENC Status Channel 1/Counter value
//     Enc/Inputs/In/nDataIn2 <-> ENC Status Channel 1/Latch value
//     Enc/Inputs/In/nState1 @bit 4 <-> ENC Status Channel 1/Status/Counter overflow
//     Enc/Inputs/In/nState1 @bit 3 <-> ENC Status Channel 1/Status/Counter underflow
//     Enc/Inputs/In/nState1 @bit 1 <-> ENC Status Channel 1/Status/Latch extern valid
//     Enc/Inputs/In/nState1 @bit 6 <-> ENC Status Channel 1/Status/Open circuit
//     Enc/Inputs/In/nState1 @bit 2 <-> ENC Status Channel 1/Status/Set counter done
//     Enc/Inputs/In/nState2 <-> ENC Status Channel 1/Status/Status of input A
//     Enc/Inputs/In/nState2 @bit 1 <-> ENC Status Channel 1/Status/Status of input B
//     Enc/Inputs/In/nState2 @bit 3 <-> ENC Status Channel 1/Status/Status of input gate
//     Enc/Inputs/In/nState4 @bit 1 <-> WcState/InputToggle
//     Enc/Inputs/In/nState4 <-> WcState/WcState
//     Enc/Outputs/Out/nCtrl1 @bit 3 <-> ENC Control Channel 1/Control/Enable latch extern on negative edge
//     Enc/Outputs/Out/nCtrl1 @bit 1 <-> ENC Control Channel 1/Control/Enable latch extern on positive edge
//     Enc/Outputs/Out/nCtrl1 @bit 2 <-> ENC Control Channel 1/Control/Set counter
//     Enc/Outputs/Out/nCtrl2 @bit 2 <-> ENC Control Channel 1/Control/Set counter on latch extern on negative edge
//     Enc/Outputs/Out/nCtrl2 @bit 1 <-> ENC Control Channel 1/Control/Set counter on latch extern on positive edge
//     Enc/Outputs/Out/nCtrl2 <-> ENC Control Channel 1/Control/Set software gate
//     Enc/Outputs/Out/nDataOut1 <-> ENC Control Channel 1/Set counter value
//   (this object) <-> Device 1 (EtherCAT)/Term 5 (EK1200)/Term 6 (EK1122-0080)/DRL02-EK0 (EK1101-0080)/DRL02-E25 (EL5042)
//     Enc/Inputs/In/nComState @bit 1 <-> WcState/InputToggle
//     Enc/Inputs/In/nComState <-> WcState/WcState
//     Enc/Inputs/In/nDataIn1 <-> FB Inputs Channel 2/Position
//     Enc/Inputs/In/nState1 @bit 12 <-> FB Inputs Channel 2/Status/Diag
//     Enc/Inputs/In/nState1 @bit 1 <-> FB Inputs Channel 2/Status/Error
//     Enc/Inputs/In/nState1 @bit 14 <-> FB Inputs Channel 2/Status/Input cycle counter
//     Enc/Inputs/In/nState1 @bit 2 <-> FB Inputs Channel 2/Status/Ready
//     Enc/Inputs/In/nState1 @bit 13 <-> FB Inputs Channel 2/Status/TxPDO State
//     Enc/Inputs/In/nState1 <-> FB Inputs Channel 2/Status/Warning
//   (this object) <-> Device 1 (EtherCAT)/Term 5 (EK1200)/Term 6 (EK1122-0080)/DRL02-EK0 (EK1101-0080)/DRL02-E26 (EL7031)
//     Drive/Inputs/In/nState1 @bit 3 <-> STM Status/Status/Error
//     Drive/Inputs/In/nState1 @bit 5 <-> STM Status/Status/Moving negative
//     Drive/Inputs/In/nState1 @bit 4 <-> STM Status/Status/Moving positive
//     Drive/Inputs/In/nState1 @bit 1 <-> STM Status/Status/Ready
//     Drive/Inputs/In/nState1 <-> STM Status/Status/Ready to enable
//     Drive/Inputs/In/nState1 @bit 6 <-> STM Status/Status/Torque reduced
//     Drive/Inputs/In/nState1 @bit 2 <-> STM Status/Status/Warning
//     Drive/Inputs/In/nState2 @bit 3 <-> STM Status/Status/Digital input 1
//     Drive/Inputs/In/nState2 @bit 4 <-> STM Status/Status/Digital input 2
//     Drive/Inputs/In/nState2 @bit 5 <-> STM Status/Status/Sync error
//     Drive/Inputs/In/nState2 @bit 7 <-> STM Status/Status/TxPDO Toggle
//     Drive/Inputs/In/nState4 @bit 1 <-> WcState/InputToggle
//     Drive/Inputs/In/nState4 <-> WcState/WcState
//     Drive/Outputs/Out/nCtrl1 <-> STM Control/Control/Enable
//     Drive/Outputs/Out/nCtrl1 @bit 2 <-> STM Control/Control/Reduce torque
//     Drive/Outputs/Out/nCtrl1 @bit 1 <-> STM Control/Control/Reset
//     Drive/Outputs/Out/nDataOut2[0] <-> STM Velocity/Velocity
//   (this object) <-> Device 1 (EtherCAT)/Term 5 (EK1200)/Term 6 (EK1122-0080)/DRL02-EK0 (EK1101-0080)/DRL02-E27 (EL7031)
//     Drive/Inputs/In/nState1 @bit 3 <-> STM Status/Status/Error
//     Drive/Inputs/In/nState1 @bit 5 <-> STM Status/Status/Moving negative
//     Drive/Inputs/In/nState1 @bit 4 <-> STM Status/Status/Moving positive
//     Drive/Inputs/In/nState1 @bit 1 <-> STM Status/Status/Ready
//     Drive/Inputs/In/nState1 <-> STM Status/Status/Ready to enable
//     Drive/Inputs/In/nState1 @bit 6 <-> STM Status/Status/Torque reduced
//     Drive/Inputs/In/nState1 @bit 2 <-> STM Status/Status/Warning
//     Drive/Inputs/In/nState2 @bit 3 <-> STM Status/Status/Digital input 1
//     Drive/Inputs/In/nState2 @bit 4 <-> STM Status/Status/Digital input 2
//     Drive/Inputs/In/nState2 @bit 5 <-> STM Status/Status/Sync error
//     Drive/Inputs/In/nState2 @bit 7 <-> STM Status/Status/TxPDO Toggle
//     Drive/Inputs/In/nState4 @bit 1 <-> WcState/InputToggle
//     Drive/Inputs/In/nState4 <-> WcState/WcState
//     Drive/Outputs/Out/nCtrl1 <-> STM Control/Control/Enable
//     Drive/Outputs/Out/nCtrl1 @bit 2 <-> STM Control/Control/Reduce torque
//     Drive/Outputs/Out/nCtrl1 @bit 1 <-> STM Control/Control/Reset
//     Drive/Outputs/Out/nDataOut2[0] <-> STM Velocity/Velocity
//     Enc/Inputs/In/nDataIn1[0] <-> ENC Status compact/Counter value
//     Enc/Inputs/In/nDataIn2[0] <-> ENC Status compact/Latch value
//     Enc/Inputs/In/nState1 @bit 4 <-> ENC Status compact/Status/Counter overflow
//     Enc/Inputs/In/nState1 @bit 3 <-> ENC Status compact/Status/Counter underflow
//     Enc/Inputs/In/nState1 @bit 1 <-> ENC Status compact/Status/Latch extern valid
//     Enc/Inputs/In/nState1 @bit 2 <-> ENC Status compact/Status/Set counter done
//     Enc/Inputs/In/nState2 @bit 4 <-> ENC Status compact/Status/Status of extern latch
//     Enc/Inputs/In/nState2 @bit 5 <-> ENC Status compact/Status/Sync error
//     Enc/Inputs/In/nState2 @bit 7 <-> ENC Status compact/Status/TxPDO Toggle
//     Enc/Inputs/In/nState4 @bit 1 <-> WcState/InputToggle
//     Enc/Inputs/In/nState4 <-> WcState/WcState
//     Enc/Outputs/Out/nCtrl1 @bit 3 <-> ENC Control compact/Control/Enable latch extern on negative edge
//     Enc/Outputs/Out/nCtrl1 @bit 1 <-> ENC Control compact/Control/Enable latch extern on positive edge
//     Enc/Outputs/Out/nCtrl1 @bit 2 <-> ENC Control compact/Control/Set counter
//     Enc/Outputs/Out/nDataOut1[0] <-> ENC Control compact/Set counter value
//   (this object) <-> Device 1 (EtherCAT)/Term 5 (EK1200)/Term 6 (EK1122-0080)/DRL02-EK0 (EK1101-0080)/DRL02-E29 (EL7031)
//     Drive/Inputs/In/nState1 @bit 3 <-> STM Status/Status/Error
//     Drive/Inputs/In/nState1 @bit 5 <-> STM Status/Status/Moving negative
//     Drive/Inputs/In/nState1 @bit 4 <-> STM Status/Status/Moving positive
//     Drive/Inputs/In/nState1 @bit 1 <-> STM Status/Status/Ready
//     Drive/Inputs/In/nState1 <-> STM Status/Status/Ready to enable
//     Drive/Inputs/In/nState1 @bit 6 <-> STM Status/Status/Torque reduced
//     Drive/Inputs/In/nState1 @bit 2 <-> STM Status/Status/Warning
//     Drive/Inputs/In/nState2 @bit 3 <-> STM Status/Status/Digital input 1
//     Drive/Inputs/In/nState2 @bit 4 <-> STM Status/Status/Digital input 2
//     Drive/Inputs/In/nState2 @bit 5 <-> STM Status/Status/Sync error
//     Drive/Inputs/In/nState2 @bit 7 <-> STM Status/Status/TxPDO Toggle
//     Drive/Inputs/In/nState4 @bit 1 <-> WcState/InputToggle
//     Drive/Inputs/In/nState4 <-> WcState/WcState
//     Drive/Outputs/Out/nCtrl1 <-> STM Control/Control/Enable
//     Drive/Outputs/Out/nCtrl1 @bit 2 <-> STM Control/Control/Reduce torque
//     Drive/Outputs/Out/nCtrl1 @bit 1 <-> STM Control/Control/Reset
//     Drive/Outputs/Out/nDataOut2[0] <-> STM Velocity/Velocity
//     Enc/Inputs/In/nDataIn1[0] <-> ENC Status compact/Counter value
//     Enc/Inputs/In/nDataIn2[0] <-> ENC Status compact/Latch value
//     Enc/Inputs/In/nState1 @bit 4 <-> ENC Status compact/Status/Counter overflow
//     Enc/Inputs/In/nState1 @bit 3 <-> ENC Status compact/Status/Counter underflow
//     Enc/Inputs/In/nState1 @bit 1 <-> ENC Status compact/Status/Latch extern valid
//     Enc/Inputs/In/nState1 @bit 2 <-> ENC Status compact/Status/Set counter done
//     Enc/Inputs/In/nState2 @bit 4 <-> ENC Status compact/Status/Status of extern latch
//     Enc/Inputs/In/nState2 @bit 5 <-> ENC Status compact/Status/Sync error
//     Enc/Inputs/In/nState2 @bit 7 <-> ENC Status compact/Status/TxPDO Toggle
//     Enc/Inputs/In/nState4 @bit 1 <-> WcState/InputToggle
//     Enc/Inputs/In/nState4 <-> WcState/WcState
//     Enc/Outputs/Out/nCtrl1 @bit 3 <-> ENC Control compact/Control/Enable latch extern on negative edge
//     Enc/Outputs/Out/nCtrl1 @bit 1 <-> ENC Control compact/Control/Enable latch extern on positive edge
//     Enc/Outputs/Out/nCtrl1 @bit 2 <-> ENC Control compact/Control/Set counter
//     Enc/Outputs/Out/nDataOut1[0] <-> ENC Control compact/Set counter value
//   (this object) <-> Device 1 (EtherCAT)/Term 5 (EK1200)/Term 6 (EK1122-0080)/DRL02-EK0 (EK1101-0080)/DRL02-E30 (EL7031)
//     Drive/Inputs/In/nState1 @bit 3 <-> STM Status/Status/Error
//     Drive/Inputs/In/nState1 @bit 5 <-> STM Status/Status/Moving negative
//     Drive/Inputs/In/nState1 @bit 4 <-> STM Status/Status/Moving positive
//     Drive/Inputs/In/nState1 @bit 1 <-> STM Status/Status/Ready
//     Drive/Inputs/In/nState1 <-> STM Status/Status/Ready to enable
//     Drive/Inputs/In/nState1 @bit 6 <-> STM Status/Status/Torque reduced
//     Drive/Inputs/In/nState1 @bit 2 <-> STM Status/Status/Warning
//     Drive/Inputs/In/nState2 @bit 3 <-> STM Status/Status/Digital input 1
//     Drive/Inputs/In/nState2 @bit 4 <-> STM Status/Status/Digital input 2
//     Drive/Inputs/In/nState2 @bit 5 <-> STM Status/Status/Sync error
//     Drive/Inputs/In/nState2 @bit 7 <-> STM Status/Status/TxPDO Toggle
//     Drive/Inputs/In/nState4 @bit 1 <-> WcState/InputToggle
//     Drive/Inputs/In/nState4 <-> WcState/WcState
//     Drive/Outputs/Out/nCtrl1 <-> STM Control/Control/Enable
//     Drive/Outputs/Out/nCtrl1 @bit 2 <-> STM Control/Control/Reduce torque
//     Drive/Outputs/Out/nCtrl1 @bit 1 <-> STM Control/Control/Reset
//     Drive/Outputs/Out/nDataOut2[0] <-> STM Velocity/Velocity
//     Enc/Inputs/In/nDataIn1[0] <-> ENC Status compact/Counter value
//     Enc/Inputs/In/nDataIn2[0] <-> ENC Status compact/Latch value
//     Enc/Inputs/In/nState1 @bit 4 <-> ENC Status compact/Status/Counter overflow
//     Enc/Inputs/In/nState1 @bit 3 <-> ENC Status compact/Status/Counter underflow
//     Enc/Inputs/In/nState1 @bit 1 <-> ENC Status compact/Status/Latch extern valid
//     Enc/Inputs/In/nState1 @bit 2 <-> ENC Status compact/Status/Set counter done
//     Enc/Inputs/In/nState2 @bit 4 <-> ENC Status compact/Status/Status of extern latch
//     Enc/Inputs/In/nState2 @bit 5 <-> ENC Status compact/Status/Sync error
//     Enc/Inputs/In/nState2 @bit 7 <-> ENC Status compact/Status/TxPDO Toggle
//     Enc/Inputs/In/nState4 @bit 1 <-> WcState/InputToggle
//     Enc/Inputs/In/nState4 <-> WcState/WcState
//     Enc/Outputs/Out/nCtrl1 @bit 3 <-> ENC Control compact/Control/Enable latch extern on negative edge
//     Enc/Outputs/Out/nCtrl1 @bit 1 <-> ENC Control compact/Control/Enable latch extern on positive edge
//     Enc/Outputs/Out/nCtrl1 @bit 2 <-> ENC Control compact/Control/Set counter
//     Enc/Outputs/Out/nDataOut1[0] <-> ENC Control compact/Set counter value
//   (this object) <-> Device 1 (EtherCAT)/Term 5 (EK1200)/Term 6 (EK1122-0080)/DRL02-EK0 (EK1101-0080)/DRL02-E33 (EL7031)
//     Drive/Inputs/In/nState1 @bit 3 <-> STM Status/Status/Error
//     Drive/Inputs/In/nState1 @bit 5 <-> STM Status/Status/Moving negative
//     Drive/Inputs/In/nState1 @bit 4 <-> STM Status/Status/Moving positive
//     Drive/Inputs/In/nState1 @bit 1 <-> STM Status/Status/Ready
//     Drive/Inputs/In/nState1 <-> STM Status/Status/Ready to enable
//     Drive/Inputs/In/nState1 @bit 6 <-> STM Status/Status/Torque reduced
//     Drive/Inputs/In/nState1 @bit 2 <-> STM Status/Status/Warning
//     Drive/Inputs/In/nState2 @bit 3 <-> STM Status/Status/Digital input 1
//     Drive/Inputs/In/nState2 @bit 4 <-> STM Status/Status/Digital input 2
//     Drive/Inputs/In/nState2 @bit 5 <-> STM Status/Status/Sync error
//     Drive/Inputs/In/nState2 @bit 7 <-> STM Status/Status/TxPDO Toggle
//     Drive/Inputs/In/nState4 @bit 1 <-> WcState/InputToggle
//     Drive/Inputs/In/nState4 <-> WcState/WcState
//     Drive/Outputs/Out/nCtrl1 <-> STM Control/Control/Enable
//     Drive/Outputs/Out/nCtrl1 @bit 2 <-> STM Control/Control/Reduce torque
//     Drive/Outputs/Out/nCtrl1 @bit 1 <-> STM Control/Control/Reset
//     Drive/Outputs/Out/nDataOut2[0] <-> STM Velocity/Velocity
//   (this object) <-> Device 1 (EtherCAT)/Term 5 (EK1200)/Term 6 (EK1122-0080)/DRL02-EK0 (EK1101-0080)/DRL02-E31 (EL7031)
//     Drive/Inputs/In/nState1 @bit 3 <-> STM Status/Status/Error
//     Drive/Inputs/In/nState1 @bit 5 <-> STM Status/Status/Moving negative
//     Drive/Inputs/In/nState1 @bit 4 <-> STM Status/Status/Moving positive
//     Drive/Inputs/In/nState1 @bit 1 <-> STM Status/Status/Ready
//     Drive/Inputs/In/nState1 <-> STM Status/Status/Ready to enable
//     Drive/Inputs/In/nState1 @bit 6 <-> STM Status/Status/Torque reduced
//     Drive/Inputs/In/nState1 @bit 2 <-> STM Status/Status/Warning
//     Drive/Inputs/In/nState2 @bit 3 <-> STM Status/Status/Digital input 1
//     Drive/Inputs/In/nState2 @bit 4 <-> STM Status/Status/Digital input 2
//     Drive/Inputs/In/nState2 @bit 5 <-> STM Status/Status/Sync error
//     Drive/Inputs/In/nState2 @bit 7 <-> STM Status/Status/TxPDO Toggle
//     Drive/Inputs/In/nState4 @bit 1 <-> WcState/InputToggle
//     Drive/Inputs/In/nState4 <-> WcState/WcState
//     Drive/Outputs/Out/nCtrl1 <-> STM Control/Control/Enable
//     Drive/Outputs/Out/nCtrl1 @bit 2 <-> STM Control/Control/Reduce torque
//     Drive/Outputs/Out/nCtrl1 @bit 1 <-> STM Control/Control/Reset
//     Drive/Outputs/Out/nDataOut2[0] <-> STM Velocity/Velocity
//   (this object) <-> Device 1 (EtherCAT)/Term 5 (EK1200)/Term 6 (EK1122-0080)/DRL02-EK0 (EK1101-0080)/DRL02-E32 (EL5042)
//     Enc/Inputs/In/nComState @bit 1 <-> WcState/InputToggle
//     Enc/Inputs/In/nComState <-> WcState/WcState
//     Enc/Inputs/In/nDataIn1 <-> FB Inputs Channel 1/Position
//     Enc/Inputs/In/nState1 @bit 12 <-> FB Inputs Channel 1/Status/Diag
//     Enc/Inputs/In/nState1 @bit 1 <-> FB Inputs Channel 1/Status/Error
//     Enc/Inputs/In/nState1 @bit 14 <-> FB Inputs Channel 1/Status/Input cycle counter
//     Enc/Inputs/In/nState1 @bit 2 <-> FB Inputs Channel 1/Status/Ready
//     Enc/Inputs/In/nState1 @bit 13 <-> FB Inputs Channel 1/Status/TxPDO State
//     Enc/Inputs/In/nState1 <-> FB Inputs Channel 1/Status/Warning
//   (this object) <-> Device 1 (EtherCAT)/Term 5 (EK1200)/Term 6 (EK1122-0080)/DRL02-EK0 (EK1101-0080)/DRL02-E28 (EL5042)
//     Enc/Inputs/In/nComState @bit 1 <-> WcState/InputToggle
//     Enc/Inputs/In/nComState <-> WcState/WcState
//     Enc/Inputs/In/nDataIn1 <-> FB Inputs Channel 1/Position
//     Enc/Inputs/In/nState1 @bit 12 <-> FB Inputs Channel 1/Status/Diag
//     Enc/Inputs/In/nState1 @bit 1 <-> FB Inputs Channel 1/Status/Error
//     Enc/Inputs/In/nState1 @bit 14 <-> FB Inputs Channel 1/Status/Input cycle counter
//     Enc/Inputs/In/nState1 @bit 2 <-> FB Inputs Channel 1/Status/Ready
//     Enc/Inputs/In/nState1 @bit 13 <-> FB Inputs Channel 1/Status/TxPDO State
//     Enc/Inputs/In/nState1 <-> FB Inputs Channel 1/Status/Warning
//   PLC_CRIX_MOT Instance <-> Device 1 (EtherCAT)/Term 5 (EK1200)/Term 167 (EK1122)/CRIX_VAC_INTF (EL6695-0002)
//     PlcTask Inputs/PRG_CryoPump.bCRYO_VGC_01_CLS <-> IO Inputs/bCRYO_VGC_01_CLS
//     PlcTask Inputs/PRG_CryoPump.bCRYO_VGC_02_CLS <-> IO Inputs/bCRYO_VGC_02_CLS
//     PlcTask Inputs/PRG_CryoPump.bCRYO_VGC_01_OPN <-> IO Inputs/bCRYO_VGC_01_OPN
//     PlcTask Inputs/PRG_CryoPump.bCRYO_VGC_02_OPN <-> IO Inputs/bCRYO_VGC_02_OPN
//     PlcTask Inputs/PRG_CryoPump.xEcatBridge_TxPDO_state <-> SYNC Inputs/TxPDO state
//     PlcTask Inputs/PRG_CryoPump.xEcatBridge_WcState <-> WcState/WcState
//     PlcTask Inputs/PRG_InjectorMotors.bSDS_VGC_01_CLS <-> IO Inputs/bSDS_VGC_01_CLS
//     PlcTask Inputs/PRG_InjectorMotors.bSDS_VGC_01_OPN <-> IO Inputs/bSDS_VGC_01_OPN
//     PlcTask Outputs/PRG_CryoPump.bMOTY10_IN <-> IO Outputs/bMOTY10_IN
//     PlcTask Outputs/PRG_CryoPump.bMOTY11_IN <-> IO Outputs/bMOTY11_IN
//     PlcTask Outputs/PRG_CryoPump.bMOTY10_OUT <-> IO Outputs/bMOTY10_OUT
//     PlcTask Outputs/PRG_CryoPump.bMOTY11_OUT <-> IO Outputs/bMOTY11_OUT
//     PlcTask Outputs/PRG_InjectorMotors.bMOTSDSZ18_IN <-> IO Outputs/bMOTSDSZ18_IN
//     PlcTask Outputs/PRG_InjectorMotors.bMOTSDSZ18_OUT <-> IO Outputs/bMOTSDSZ18_OUT
//   PLC_CRIX_MOT Instance <-> Device 1 (EtherCAT)/Term 5 (EK1200)/Term 6 (EK1122-0080)/DRL02-EK0 (EK1101-0080)/DRL02-E1 (EL7031)
//     PlcTask Inputs/Main.M1.bLimitBackwardEnable <-> STM Status/Status/Digital input 1
//     PlcTask Inputs/Main.M1.bLimitForwardEnable <-> STM Status/Status/Digital input 2
//   PLC_CRIX_MOT Instance <-> Device 1 (EtherCAT)/Term 5 (EK1200)/Term 6 (EK1122-0080)/DRL02-EK0 (EK1101-0080)/DRL02-E11 (EL7031)
//     PlcTask Inputs/Main.M7.bLimitBackwardEnable <-> STM Status/Status/Digital input 2
//     PlcTask Inputs/Main.M7.bLimitForwardEnable <-> STM Status/Status/Digital input 1
//   PLC_CRIX_MOT Instance <-> Device 1 (EtherCAT)/Term 5 (EK1200)/Term 6 (EK1122-0080)/DRL02-EK0 (EK1101-0080)/DRL02-E13 (EL7041)
//     PlcTask Inputs/Main.M8.bLimitBackwardEnable <-> STM Status/Status/Digital input 2
//     PlcTask Inputs/Main.M8.bLimitForwardEnable <-> STM Status/Status/Digital input 1
//   PLC_CRIX_MOT Instance <-> Device 1 (EtherCAT)/Term 5 (EK1200)/Term 6 (EK1122-0080)/DRL02-EK0 (EK1101-0080)/DRL02-E17 (EL7031)
//     PlcTask Inputs/Main.M12.bLimitBackwardEnable <-> STM Status/Status/Digital input 2
//     PlcTask Inputs/Main.M12.bLimitForwardEnable <-> STM Status/Status/Digital input 1
//   PLC_CRIX_MOT Instance <-> Device 1 (EtherCAT)/Term 5 (EK1200)/Term 6 (EK1122-0080)/DRL02-EK0 (EK1101-0080)/DRL02-E19 (EL7031)
//     PlcTask Inputs/Main.M13.bLimitBackwardEnable <-> STM Status/Status/Digital input 2
//     PlcTask Inputs/Main.M13.bLimitForwardEnable <-> STM Status/Status/Digital input 1
//   PLC_CRIX_MOT Instance <-> Device 1 (EtherCAT)/Term 5 (EK1200)/Term 6 (EK1122-0080)/DRL02-EK0 (EK1101-0080)/DRL02-E21 (EL7041)
//     PlcTask Inputs/Main.M49.bLimitForwardEnable <-> STM Status/Status/Digital input 2
//     PlcTask Inputs/PRG_CryoPump.bLimitBackwardEnable_Y_11 <-> STM Status/Status/Digital input 1
//   PLC_CRIX_MOT Instance <-> Device 1 (EtherCAT)/Term 5 (EK1200)/Term 6 (EK1122-0080)/DRL02-EK0 (EK1101-0080)/DRL02-E23 (EL7041)
//     PlcTask Inputs/Main.M48.bLimitForwardEnable <-> STM Status/Status/Digital input 2
//     PlcTask Inputs/PRG_CryoPump.bLimitBackwardEnable_Y_10 <-> STM Status/Status/Digital input 1
//   PLC_CRIX_MOT Instance <-> Device 1 (EtherCAT)/Term 5 (EK1200)/Term 6 (EK1122-0080)/DRL02-EK0 (EK1101-0080)/DRL02-E26 (EL7031)
//     PlcTask Inputs/Main.M17.bLimitBackwardEnable <-> STM Status/Status/Digital input 2
//     PlcTask Inputs/Main.M17.bLimitForwardEnable <-> STM Status/Status/Digital input 1
//   PLC_CRIX_MOT Instance <-> Device 1 (EtherCAT)/Term 5 (EK1200)/Term 6 (EK1122-0080)/DRL02-EK0 (EK1101-0080)/DRL02-E27 (EL7031)
//     PlcTask Inputs/Main.M18.bLimitForwardEnable <-> STM Status/Status/Digital input 1
//     PlcTask Inputs/PRG_InjectorMotors.bLimitBackwardEnable_SDSZ_18 <-> STM Status/Status/Digital input 2
//   PLC_CRIX_MOT Instance <-> Device 1 (EtherCAT)/Term 5 (EK1200)/Term 6 (EK1122-0080)/DRL02-EK0 (EK1101-0080)/DRL02-E3 (EL7031)
//     PlcTask Inputs/Main.M2.bLimitBackwardEnable <-> STM Status/Status/Digital input 2
//     PlcTask Inputs/Main.M2.bLimitForwardEnable <-> STM Status/Status/Digital input 1
//   PLC_CRIX_MOT Instance <-> Device 1 (EtherCAT)/Term 5 (EK1200)/Term 6 (EK1122-0080)/DRL02-EK0 (EK1101-0080)/DRL02-E31 (EL7031)
//     PlcTask Inputs/Main.M35.bLimitBackwardEnable <-> STM Status/Status/Digital input 2
//     PlcTask Inputs/Main.M35.bLimitForwardEnable <-> STM Status/Status/Digital input 1
//   PLC_CRIX_MOT Instance <-> Device 1 (EtherCAT)/Term 5 (EK1200)/Term 6 (EK1122-0080)/DRL02-EK0 (EK1101-0080)/DRL02-E4 (EL7031)
//     PlcTask Inputs/Main.M3.bLimitBackwardEnable <-> STM Status/Status/Digital input 2
//     PlcTask Inputs/Main.M3.bLimitForwardEnable <-> STM Status/Status/Digital input 1
//   PLC_CRIX_MOT Instance <-> Device 1 (EtherCAT)/Term 5 (EK1200)/Term 6 (EK1122-0080)/DRL02-EK0 (EK1101-0080)/DRL02-E6 (EL7031)
//     PlcTask Inputs/Main.M4.bLimitBackwardEnable <-> STM Status/Status/Digital input 1
//     PlcTask Inputs/Main.M4.bLimitForwardEnable <-> STM Status/Status/Digital input 2
//   PLC_CRIX_MOT Instance <-> Device 1 (EtherCAT)/Term 5 (EK1200)/Term 6 (EK1122-0080)/DRL02-EK0 (EK1101-0080)/DRL02-E7 (EL7031)
//     PlcTask Inputs/Main.M5.bLimitBackwardEnable <-> STM Status/Status/Digital input 2
//     PlcTask Inputs/Main.M5.bLimitForwardEnable <-> STM Status/Status/Digital input 1
//   PLC_CRIX_MOT Instance <-> Device 1 (EtherCAT)/Term 5 (EK1200)/Term 6 (EK1122-0080)/DRL02-EK0 (EK1101-0080)/DRL02-E9 (EL7031)
//     PlcTask Inputs/Main.M6.bLimitBackwardEnable <-> STM Status/Status/Digital input 2
//     PlcTask Inputs/Main.M6.bLimitForwardEnable <-> STM Status/Status/Digital input 1
//   PLC_CRIX_MOT Instance <-> Device 1 (EtherCAT)/Term 5 (EK1200)/Term 6 (EK1122-0080)/DRL02-EK0 (EK1101-0080)/DRL02-ECJ0 (EK1122-0080)/Term 109 (EK1101-0080)/Camera X (EL7041)
//     PlcTask Inputs/Main.M33.bLimitBackwardEnable <-> STM Status/Status/Digital input 2
//     PlcTask Inputs/Main.M33.bLimitForwardEnable <-> STM Status/Status/Digital input 1
//   PLC_CRIX_MOT Instance <-> Device 1 (EtherCAT)/Term 5 (EK1200)/Term 6 (EK1122-0080)/DRL02-EK0 (EK1101-0080)/DRL02-ECJ0 (EK1122-0080)/Term 109 (EK1101-0080)/Camera Y (EL7041)
//     PlcTask Inputs/Main.M34.bLimitBackwardEnable <-> STM Status/Status/Digital input 2
//     PlcTask Inputs/Main.M34.bLimitForwardEnable <-> STM Status/Status/Digital input 1
//   PLC_CRIX_MOT Instance <-> Device 1 (EtherCAT)/Term 5 (EK1200)/Term 6 (EK1122-0080)/DRL02-EK0 (EK1101-0080)/DRL02-ECJ0 (EK1122-0080)/Term 113 (EK1101-0080)/Beamblock X (EL7041)
//     PlcTask Inputs/Main.M30.bLimitBackwardEnable <-> STM Status/Status/Digital input 2
//     PlcTask Inputs/Main.M30.bLimitForwardEnable <-> STM Status/Status/Digital input 1
//   PLC_CRIX_MOT Instance <-> Device 1 (EtherCAT)/Term 5 (EK1200)/Term 6 (EK1122-0080)/DRL02-EK0 (EK1101-0080)/DRL02-ECJ0 (EK1122-0080)/Term 113 (EK1101-0080)/Beamblock Y (EL7041)
//     PlcTask Inputs/Main.M31.bLimitBackwardEnable <-> STM Status/Status/Digital input 2
//     PlcTask Inputs/Main.M31.bLimitForwardEnable <-> STM Status/Status/Digital input 1
//   PLC_CRIX_MOT Instance <-> Device 1 (EtherCAT)/Term 5 (EK1200)/Term 6 (EK1122-0080)/DRL02-EK0 (EK1101-0080)/DRL02-ECJ0 (EK1122-0080)/Term 113 (EK1101-0080)/Beamblock Z (EL7041)
//     PlcTask Inputs/Main.M32.bLimitBackwardEnable <-> STM Status/Status/Digital input 2
//     PlcTask Inputs/Main.M32.bLimitForwardEnable <-> STM Status/Status/Digital input 1
//   PLC_CRIX_MOT Instance <-> Device 1 (EtherCAT)/Term 5 (EK1200)/Term 6 (EK1122-0080)/DRL02-EK0 (EK1101-0080)/DRL02-ECJ1 (EK1122)/CryoStat (EK1101)/Cryo X (EL7041)
//     PlcTask Inputs/Main.M22.bLimitBackwardEnable <-> STM Status/Status/Digital input 2
//     PlcTask Inputs/Main.M22.bLimitForwardEnable <-> STM Status/Status/Digital input 1
//   PLC_CRIX_MOT Instance <-> Device 1 (EtherCAT)/Term 5 (EK1200)/Term 6 (EK1122-0080)/DRL02-EK0 (EK1101-0080)/DRL02-ECJ1 (EK1122)/CryoStat (EK1101)/Cryo Y (EL7041)
//     PlcTask Inputs/Main.M23.bLimitBackwardEnable <-> STM Status/Status/Digital input 2
//     PlcTask Inputs/Main.M23.bLimitForwardEnable <-> STM Status/Status/Digital input 1
//   PLC_CRIX_MOT Instance <-> Device 1 (EtherCAT)/Term 5 (EK1200)/Term 6 (EK1122-0080)/DRL02-EK0 (EK1101-0080)/DRL02-ECJ1 (EK1122)/CryoStat (EK1101)/Cryo Z (EL7041)
//     PlcTask Inputs/Main.M24.bLimitBackwardEnable <-> STM Status/Status/Digital input 2
//     PlcTask Inputs/Main.M24.bLimitForwardEnable <-> STM Status/Status/Digital input 1
//   PLC_CRIX_MOT Instance <-> Device 1 (EtherCAT)/Term 5 (EK1200)/Term 6 (EK1122-0080)/DRL02-EK0 (EK1101-0080)/DRL02-ECJ1 (EK1122)/CryoStat (EK1101)/Term 158 (EL4004)
//     PlcTask Outputs/GVL_FiberLite.bLedOutput1.iIlluminatorINT <-> AO Outputs Channel 1/Analog output
//   PLC_CRIX_MOT Instance <-> Device 1 (EtherCAT)/Term 5 (EK1200)/Term 6 (EK1122-0080)/DRL02-EK0 (EK1101-0080)/DRL02-ECJ1 (EK1122)/VLS_EP10_EP7041-3102
//     PlcTask Inputs/Main.M44.bHome <-> ENC Status compact/Status/Status of input C
//     PlcTask Inputs/Main.M44.bLimitBackwardEnable <-> STM Status/Status/Digital input 1
//     PlcTask Inputs/Main.M44.bLimitForwardEnable <-> STM Status/Status/Digital input 2
//     PlcTask Inputs/Main.M44.nRawEncoderUINT <-> ENC Status compact/Counter value
//   PLC_CRIX_MOT Instance <-> Device 1 (EtherCAT)/Term 5 (EK1200)/Term 6 (EK1122-0080)/DRL02-EK0 (EK1101-0080)/DRL02-ECJ1 (EK1122)/VLS_EP11_EP7041-3102
//     PlcTask Inputs/Main.M45.bHome <-> ENC Status compact/Status/Status of input C
//     PlcTask Inputs/Main.M45.bLimitBackwardEnable <-> STM Status/Status/Digital input 1
//     PlcTask Inputs/Main.M45.bLimitForwardEnable <-> STM Status/Status/Digital input 2
//     PlcTask Inputs/Main.M45.nRawEncoderUINT <-> ENC Status compact/Counter value
//   PLC_CRIX_MOT Instance <-> Device 1 (EtherCAT)/Term 5 (EK1200)/Term 6 (EK1122-0080)/DRL02-EK0 (EK1101-0080)/DRL02-ECJ1 (EK1122)/VLS_EP12_EP7041-3102
//     PlcTask Inputs/Main.M46.bHome <-> ENC Status compact/Status/Status of input C
//     PlcTask Inputs/Main.M46.bLimitBackwardEnable <-> STM Status/Status/Digital input 2
//     PlcTask Inputs/Main.M46.bLimitForwardEnable <-> STM Status/Status/Digital input 1
//   PLC_CRIX_MOT Instance <-> Device 1 (EtherCAT)/Term 5 (EK1200)/Term 6 (EK1122-0080)/DRL02-EK0 (EK1101-0080)/DRL02-ECJ1 (EK1122)/VLS_EP13_EP7041-3102
//     PlcTask Inputs/Main.M47.bHome <-> ENC Status compact/Status/Status of input C
//     PlcTask Inputs/Main.M47.bLimitBackwardEnable <-> STM Status/Status/Digital input 1
//     PlcTask Inputs/Main.M47.bLimitForwardEnable <-> STM Status/Status/Digital input 2
//   PLC_CRIX_MOT Instance <-> Device 1 (EtherCAT)/Term 5 (EK1200)/Term 6 (EK1122-0080)/DRL02-EK0 (EK1101-0080)/DRL02-ECJ1 (EK1122)/VLS_EP6_EP7041-1002
//     PlcTask Inputs/Main.M40.bLimitBackwardEnable <-> STM Status/Status/Digital input 2
//     PlcTask Inputs/Main.M40.bLimitForwardEnable <-> STM Status/Status/Digital input 1
//   PLC_CRIX_MOT Instance <-> Device 1 (EtherCAT)/Term 5 (EK1200)/Term 6 (EK1122-0080)/DRL02-EK0 (EK1101-0080)/DRL02-ECJ1 (EK1122)/VLS_EP7_EP7041-1002
//     PlcTask Inputs/Main.M41.bLimitBackwardEnable <-> STM Status/Status/Digital input 2
//     PlcTask Inputs/Main.M41.bLimitForwardEnable <-> STM Status/Status/Digital input 1
//   PLC_CRIX_MOT Instance <-> Device 1 (EtherCAT)/Term 5 (EK1200)/Term 6 (EK1122-0080)/DRL02-EK0 (EK1101-0080)/DRL02-ECJ1 (EK1122)/VLS_EP8_EP7041-1002
//     PlcTask Inputs/Main.M42.bLimitBackwardEnable <-> STM Status/Status/Digital input 2
//     PlcTask Inputs/Main.M42.bLimitForwardEnable <-> STM Status/Status/Digital input 1
//   PLC_CRIX_MOT Instance <-> Device 1 (EtherCAT)/Term 5 (EK1200)/Term 6 (EK1122-0080)/DRL02-EK0 (EK1101-0080)/DRL02-ECJ1 (EK1122)/VLS_EP9_EP7041-1002
//     PlcTask Inputs/Main.M43.bLimitBackwardEnable <-> STM Status/Status/Digital input 2
//     PlcTask Inputs/Main.M43.bLimitForwardEnable <-> STM Status/Status/Digital input 1
//   PLC_CRIX_MOT Instance <-> Device 1 (EtherCAT)/Term 5 (EK1200)/Term 6 (EK1122-0080)/DRL02-EK0 (EK1101-0080)/DRL02-ECJ2 (EK1122)/Catcher (EK1100)/Catcher_E1_EL7041
//     PlcTask Inputs/Main.M37.bLimitBackwardEnable <-> STM Status/Status/Digital input 1
//     PlcTask Inputs/Main.M37.bLimitForwardEnable <-> STM Status/Status/Digital input 2
//   PLC_CRIX_MOT Instance <-> Device 1 (EtherCAT)/Term 5 (EK1200)/Term 6 (EK1122-0080)/DRL02-EK0 (EK1101-0080)/DRL02-ECJ2 (EK1122)/Catcher (EK1100)/Catcher_E3_EL7041
//     PlcTask Inputs/Main.M38.bLimitBackwardEnable <-> STM Status/Status/Digital input 2
//     PlcTask Inputs/Main.M38.bLimitForwardEnable <-> STM Status/Status/Digital input 1
//   PLC_CRIX_MOT Instance <-> Device 1 (EtherCAT)/Term 5 (EK1200)/Term 6 (EK1122-0080)/DRL02-EK0 (EK1101-0080)/DRL02-ECJ2 (EK1122)/Catcher (EK1100)/Catcher_E4_EL7041
//     PlcTask Inputs/Main.M39.bLimitBackwardEnable <-> STM Status/Status/Digital input 1
//     PlcTask Inputs/Main.M39.bLimitForwardEnable <-> STM Status/Status/Digital input 2
//   PLC_CRIX_MOT Instance <-> Device 1 (EtherCAT)/Term 5 (EK1200)/Term 6 (EK1122-0080)/DRL02-EK0 (EK1101-0080)/Term 173 (EL1124)
//     PlcTask Inputs/PRG_InjectorMotors.bHall_Backward <-> Channel 4/Input
//     PlcTask Inputs/PRG_InjectorMotors.bHall_Forward <-> Channel 3/Input
//   PLC_CRIX_MOT Instance <-> Device 1 (EtherCAT)/Term 5 (EK1200)/Term 6 (EK1122-0080)/DRL02-EK0 (EK1101-0080)/Term 65 (EL1084)
//     PlcTask Inputs/Main.M10.bLimitBackwardEnable <-> Channel 4/Input
//     PlcTask Inputs/Main.M9.bLimitBackwardEnable <-> Channel 2/Input
//     PlcTask Inputs/Main.M10.bLimitForwardEnable <-> Channel 3/Input
//     PlcTask Inputs/Main.M9.bLimitForwardEnable <-> Channel 1/Input
//   PLC_CRIX_MOT Instance <-> Device 1 (EtherCAT)/Term 5 (EK1200)/Term 6 (EK1122-0080)/DRL02-EK0 (EK1101-0080)/Term 68 (EL1084)
//     PlcTask Inputs/Main.M11.bLimitBackwardEnable <-> Channel 2/Input
//     PlcTask Inputs/Main.M11.bLimitForwardEnable <-> Channel 1/Input
//   PLC_CRIX_MOT Instance <-> Device 1 (EtherCAT)/Term 5 (EK1200)/Term 83 (EK1521-0010)/Term 166 (EK1501-0010)/PMPS_FFO
//     PlcTask Outputs/GVL_PMPS.g_FastFaultOutput1.q_xFastFaultOut <-> Channel 1/Output
//     PlcTask Outputs/GVL_PMPS.g_FastFaultOutput2.q_xFastFaultOut <-> Channel 2/Output
//   PLC_CRIX_MOT Instance <-> Device 1 (EtherCAT)/Term 5 (EK1200)/Term 83 (EK1521-0010)/Term 166 (EK1501-0010)/PMPS_PRE
//     PlcTask Inputs/PRG_PMPS.fbArbiterIO.i_stCurrentBP <-> IO Inputs/CurrentBP
//     PlcTask Inputs/PRG_PMPS.fbArbiterIO.xTxPDO_state <-> SYNC Inputs/TxPDO state
//     PlcTask Inputs/PRG_PMPS.fbArbiterIO.xTxPDO_toggle <-> SYNC Inputs/TxPDO toggle
//     PlcTask Outputs/PRG_PMPS.fbArbiterIO.q_stRequestedBP <-> IO Outputs/RequestedBP
//   PLC_CRIX_MOT Instance <-> NC-Task 1 SAF/Axes/Axis 1 - Diagnostic Paddle X
//     PlcTask Inputs/Main.M1.Axis.NcToPlc <-> Outputs/ToPlc
//     PlcTask Outputs/Main.M1.Axis.PlcToNc <-> Inputs/FromPlc
//   PLC_CRIX_MOT Instance <-> NC-Task 1 SAF/Axes/Axis 10 - Illumination Y
//     PlcTask Inputs/Main.M10.Axis.NcToPlc <-> Outputs/ToPlc
//     PlcTask Outputs/Main.M10.Axis.PlcToNc <-> Inputs/FromPlc
//   PLC_CRIX_MOT Instance <-> NC-Task 1 SAF/Axes/Axis 11 - Illumination Z
//     PlcTask Inputs/Main.M11.Axis.NcToPlc <-> Outputs/ToPlc
//     PlcTask Outputs/Main.M11.Axis.PlcToNc <-> Inputs/FromPlc
//   PLC_CRIX_MOT Instance <-> NC-Task 1 SAF/Axes/Axis 12 - Questar X
//     PlcTask Inputs/Main.M12.Axis.NcToPlc <-> Outputs/ToPlc
//     PlcTask Outputs/Main.M12.Axis.PlcToNc <-> Inputs/FromPlc
//   PLC_CRIX_MOT Instance <-> NC-Task 1 SAF/Axes/Axis 13 - Questar Y
//     PlcTask Inputs/Main.M13.Axis.NcToPlc <-> Outputs/ToPlc
//     PlcTask Outputs/Main.M13.Axis.PlcToNc <-> Inputs/FromPlc
//   PLC_CRIX_MOT Instance <-> NC-Task 1 SAF/Axes/Axis 14 - SPARE 1
//     PlcTask Inputs/Main.M14.Axis.NcToPlc <-> Outputs/ToPlc
//     PlcTask Outputs/Main.M14.Axis.PlcToNc <-> Inputs/FromPlc
//   PLC_CRIX_MOT Instance <-> NC-Task 1 SAF/Axes/Axis 15 - SPARE 2
//     PlcTask Inputs/Main.M15.Axis.NcToPlc <-> Outputs/ToPlc
//     PlcTask Outputs/Main.M15.Axis.PlcToNc <-> Inputs/FromPlc
//   PLC_CRIX_MOT Instance <-> NC-Task 1 SAF/Axes/Axis 16 - SDS Injector X
//     PlcTask Inputs/Main.M16.Axis.NcToPlc <-> Outputs/ToPlc
//     PlcTask Outputs/Main.M16.Axis.PlcToNc <-> Inputs/FromPlc
//   PLC_CRIX_MOT Instance <-> NC-Task 1 SAF/Axes/Axis 17 - SDS Injectory Y
//     PlcTask Inputs/Main.M17.Axis.NcToPlc <-> Outputs/ToPlc
//     PlcTask Outputs/Main.M17.Axis.PlcToNc <-> Inputs/FromPlc
//   PLC_CRIX_MOT Instance <-> NC-Task 1 SAF/Axes/Axis 18 - SDS Injector Z
//     PlcTask Inputs/Main.M18.Axis.NcToPlc <-> Outputs/ToPlc
//     PlcTask Outputs/Main.M18.Axis.PlcToNc <-> Inputs/FromPlc
//   PLC_CRIX_MOT Instance <-> NC-Task 1 SAF/Axes/Axis 19 - SDS Rotation Y
//     PlcTask Inputs/Main.M19.Axis.NcToPlc <-> Outputs/ToPlc
//     PlcTask Outputs/Main.M19.Axis.PlcToNc <-> Inputs/FromPlc
//   PLC_CRIX_MOT Instance <-> NC-Task 1 SAF/Axes/Axis 2 - Diagnostic Paddle Y
//     PlcTask Inputs/Main.M2.Axis.NcToPlc <-> Outputs/ToPlc
//     PlcTask Outputs/Main.M2.Axis.PlcToNc <-> Inputs/FromPlc
//   PLC_CRIX_MOT Instance <-> NC-Task 1 SAF/Axes/Axis 20 - SDS Shroud Rotation
//     PlcTask Inputs/Main.M20.Axis.NcToPlc <-> Outputs/ToPlc
//     PlcTask Outputs/Main.M20.Axis.PlcToNc <-> Inputs/FromPlc
//   PLC_CRIX_MOT Instance <-> NC-Task 1 SAF/Axes/Axis 3 - Diagnostic Paddle Z
//     PlcTask Inputs/Main.M3.Axis.NcToPlc <-> Outputs/ToPlc
//     PlcTask Outputs/Main.M3.Axis.PlcToNc <-> Inputs/FromPlc
//   PLC_CRIX_MOT Instance <-> NC-Task 1 SAF/Axes/Axis 35 - Outcoupling Lens Y
//     PlcTask Inputs/Main.M35.Axis.NcToPlc <-> Outputs/ToPlc
//     PlcTask Outputs/Main.M35.Axis.PlcToNc <-> Inputs/FromPlc
//   PLC_CRIX_MOT Instance <-> NC-Task 1 SAF/Axes/Axis 36 - SDS Z Encoder
//     PlcTask Inputs/Main.M36.Axis.NcToPlc <-> Outputs/ToPlc
//     PlcTask Outputs/Main.M36.Axis.PlcToNc <-> Inputs/FromPlc
//   PLC_CRIX_MOT Instance <-> NC-Task 1 SAF/Axes/Axis 4 - Objectives X
//     PlcTask Inputs/Main.M4.Axis.NcToPlc <-> Outputs/ToPlc
//     PlcTask Outputs/Main.M4.Axis.PlcToNc <-> Inputs/FromPlc
//   PLC_CRIX_MOT Instance <-> NC-Task 1 SAF/Axes/Axis 5 - Objectives Y
//     PlcTask Inputs/Main.M5.Axis.NcToPlc <-> Outputs/ToPlc
//     PlcTask Outputs/Main.M5.Axis.PlcToNc <-> Inputs/FromPlc
//   PLC_CRIX_MOT Instance <-> NC-Task 1 SAF/Axes/Axis 6 - Objectives Z
//     PlcTask Inputs/Main.M6.Axis.NcToPlc <-> Outputs/ToPlc
//     PlcTask Outputs/Main.M6.Axis.PlcToNc <-> Inputs/FromPlc
//   PLC_CRIX_MOT Instance <-> NC-Task 1 SAF/Axes/Axis 7 - Point Detector Y
//     PlcTask Inputs/Main.M7.Axis.NcToPlc <-> Outputs/ToPlc
//     PlcTask Outputs/Main.M7.Axis.PlcToNc <-> Inputs/FromPlc
//   PLC_CRIX_MOT Instance <-> NC-Task 1 SAF/Axes/Axis 8 - Point Detector Rotation
//     PlcTask Inputs/Main.M8.Axis.NcToPlc <-> Outputs/ToPlc
//     PlcTask Outputs/Main.M8.Axis.PlcToNc <-> Inputs/FromPlc
//   PLC_CRIX_MOT Instance <-> NC-Task 1 SAF/Axes/Axis 9 - Illumination X
//     PlcTask Inputs/Main.M9.Axis.NcToPlc <-> Outputs/ToPlc
//     PlcTask Outputs/Main.M9.Axis.PlcToNc <-> Inputs/FromPlc
//   PLC_CRIX_MOT Instance <-> NC-Task 1 SAF/Axes/Beam X
//     PlcTask Inputs/Main.M30.Axis.NcToPlc <-> Outputs/ToPlc
//     PlcTask Outputs/Main.M30.Axis.PlcToNc <-> Inputs/FromPlc
//   PLC_CRIX_MOT Instance <-> NC-Task 1 SAF/Axes/Beam Y
//     PlcTask Inputs/Main.M31.Axis.NcToPlc <-> Outputs/ToPlc
//     PlcTask Outputs/Main.M31.Axis.PlcToNc <-> Inputs/FromPlc
//   PLC_CRIX_MOT Instance <-> NC-Task 1 SAF/Axes/Beam Z
//     PlcTask Inputs/Main.M32.Axis.NcToPlc <-> Outputs/ToPlc
//     PlcTask Outputs/Main.M32.Axis.PlcToNc <-> Inputs/FromPlc
//   PLC_CRIX_MOT Instance <-> NC-Task 1 SAF/Axes/Camera X
//     PlcTask Inputs/Main.M33.Axis.NcToPlc <-> Outputs/ToPlc
//     PlcTask Outputs/Main.M33.Axis.PlcToNc <-> Inputs/FromPlc
//   PLC_CRIX_MOT Instance <-> NC-Task 1 SAF/Axes/Camera Y
//     PlcTask Inputs/Main.M34.Axis.NcToPlc <-> Outputs/ToPlc
//     PlcTask Outputs/Main.M34.Axis.PlcToNc <-> Inputs/FromPlc
//   PLC_CRIX_MOT Instance <-> NC-Task 1 SAF/Axes/Cryo X
//     PlcTask Inputs/Main.M22.Axis.NcToPlc <-> Outputs/ToPlc
//     PlcTask Outputs/Main.M22.Axis.PlcToNc <-> Inputs/FromPlc
//   PLC_CRIX_MOT Instance <-> NC-Task 1 SAF/Axes/Cryo Y
//     PlcTask Inputs/Main.M23.Axis.NcToPlc <-> Outputs/ToPlc
//     PlcTask Outputs/Main.M23.Axis.PlcToNc <-> Inputs/FromPlc
//   PLC_CRIX_MOT Instance <-> NC-Task 1 SAF/Axes/Cryo Z
//     PlcTask Inputs/Main.M24.Axis.NcToPlc <-> Outputs/ToPlc
//     PlcTask Outputs/Main.M24.Axis.PlcToNc <-> Inputs/FromPlc
//   PLC_CRIX_MOT Instance <-> NC-Task 1 SAF/Axes/Cryo rY
//     PlcTask Inputs/Main.M25.Axis.NcToPlc <-> Outputs/ToPlc
//     PlcTask Outputs/Main.M25.Axis.PlcToNc <-> Inputs/FromPlc
//   PLC_CRIX_MOT Instance <-> NC-Task 1 SAF/Axes/M37-X
//     PlcTask Inputs/Main.M37.Axis.NcToPlc <-> Outputs/ToPlc
//     PlcTask Outputs/Main.M37.Axis.PlcToNc <-> Inputs/FromPlc
//   PLC_CRIX_MOT Instance <-> NC-Task 1 SAF/Axes/M38-Y
//     PlcTask Inputs/Main.M38.Axis.NcToPlc <-> Outputs/ToPlc
//     PlcTask Outputs/Main.M38.Axis.PlcToNc <-> Inputs/FromPlc
//   PLC_CRIX_MOT Instance <-> NC-Task 1 SAF/Axes/M39-Z
//     PlcTask Inputs/Main.M39.Axis.NcToPlc <-> Outputs/ToPlc
//     PlcTask Outputs/Main.M39.Axis.PlcToNc <-> Inputs/FromPlc
//   PLC_CRIX_MOT Instance <-> NC-Task 1 SAF/Axes/M40-VLS-Slit-Top
//     PlcTask Inputs/Main.M40.Axis.NcToPlc <-> Outputs/ToPlc
//     PlcTask Outputs/Main.M40.Axis.PlcToNc <-> Inputs/FromPlc
//   PLC_CRIX_MOT Instance <-> NC-Task 1 SAF/Axes/M41-VLS-Slit-Bottom
//     PlcTask Inputs/Main.M41.Axis.NcToPlc <-> Outputs/ToPlc
//     PlcTask Outputs/Main.M41.Axis.PlcToNc <-> Inputs/FromPlc
//   PLC_CRIX_MOT Instance <-> NC-Task 1 SAF/Axes/M42-VLS-Slit-Right
//     PlcTask Inputs/Main.M42.Axis.NcToPlc <-> Outputs/ToPlc
//     PlcTask Outputs/Main.M42.Axis.PlcToNc <-> Inputs/FromPlc
//   PLC_CRIX_MOT Instance <-> NC-Task 1 SAF/Axes/M43-VLS-Slit-Left
//     PlcTask Inputs/Main.M43.Axis.NcToPlc <-> Outputs/ToPlc
//     PlcTask Outputs/Main.M43.Axis.PlcToNc <-> Inputs/FromPlc
//   PLC_CRIX_MOT Instance <-> NC-Task 1 SAF/Axes/M44-VLS-Mirror-Pitch
//     PlcTask Inputs/Main.M44.Axis.NcToPlc <-> Outputs/ToPlc
//     PlcTask Outputs/Main.M44.Axis.PlcToNc <-> Inputs/FromPlc
//   PLC_CRIX_MOT Instance <-> NC-Task 1 SAF/Axes/M45-VLS-Grating-Pitch
//     PlcTask Inputs/Main.M45.Axis.NcToPlc <-> Outputs/ToPlc
//     PlcTask Outputs/Main.M45.Axis.PlcToNc <-> Inputs/FromPlc
//   PLC_CRIX_MOT Instance <-> NC-Task 1 SAF/Axes/M46-VLS-Camera-Pitch
//     PlcTask Inputs/Main.M46.Axis.NcToPlc <-> Outputs/ToPlc
//     PlcTask Outputs/Main.M46.Axis.PlcToNc <-> Inputs/FromPlc
//   PLC_CRIX_MOT Instance <-> NC-Task 1 SAF/Axes/M47-VLS-Camera-Dist
//     PlcTask Inputs/Main.M47.Axis.NcToPlc <-> Outputs/ToPlc
//     PlcTask Outputs/Main.M47.Axis.PlcToNc <-> Inputs/FromPlc
//   PLC_CRIX_MOT Instance <-> NC-Task 1 SAF/Axes/M48- Cryopump Y10
//     PlcTask Inputs/Main.M48.Axis.NcToPlc <-> Outputs/ToPlc
//     PlcTask Outputs/Main.M48.Axis.PlcToNc <-> Inputs/FromPlc
//   PLC_CRIX_MOT Instance <-> NC-Task 1 SAF/Axes/M49- Cryopump Y11
//     PlcTask Inputs/Main.M49.Axis.NcToPlc <-> Outputs/ToPlc
//     PlcTask Outputs/Main.M49.Axis.PlcToNc <-> Inputs/FromPlc
//   PLC_CRIX_MOT Instance <-> NC-Task 1 SAF/Axes/RCI RX
//     PlcTask Inputs/Main.M29.Axis.NcToPlc <-> Outputs/ToPlc
//     PlcTask Outputs/Main.M29.Axis.PlcToNc <-> Inputs/FromPlc
//   PLC_CRIX_MOT Instance <-> NC-Task 1 SAF/Axes/RCI X
//     PlcTask Inputs/Main.M26.Axis.NcToPlc <-> Outputs/ToPlc
//     PlcTask Outputs/Main.M26.Axis.PlcToNc <-> Inputs/FromPlc
//   PLC_CRIX_MOT Instance <-> NC-Task 1 SAF/Axes/RCI Y
//     PlcTask Inputs/Main.M27.Axis.NcToPlc <-> Outputs/ToPlc
//     PlcTask Outputs/Main.M27.Axis.PlcToNc <-> Inputs/FromPlc
//   PLC_CRIX_MOT Instance <-> NC-Task 1 SAF/Axes/RCI Z
//     PlcTask Inputs/Main.M28.Axis.NcToPlc <-> Outputs/ToPlc
//     PlcTask Outputs/Main.M28.Axis.PlcToNc <-> Inputs/FromPlc
//   PLC_CRIX_MOT Instance <-> NC-Task 1 SAF/Axes/SL2K2-BOTTOM-M50
//     PlcTask Inputs/Main.M50.Axis.NcToPlc <-> Outputs/ToPlc
//     PlcTask Outputs/Main.M50.Axis.PlcToNc <-> Inputs/FromPlc
//   PLC_CRIX_MOT Instance <-> NC-Task 1 SAF/Axes/SL2K2-NORTH-M52
//     PlcTask Inputs/Main.M52.Axis.NcToPlc <-> Outputs/ToPlc
//     PlcTask Outputs/Main.M52.Axis.PlcToNc <-> Inputs/FromPlc
//   PLC_CRIX_MOT Instance <-> NC-Task 1 SAF/Axes/SL2K2-SOUTH-M53
//     PlcTask Inputs/Main.M53.Axis.NcToPlc <-> Outputs/ToPlc
//     PlcTask Outputs/Main.M53.Axis.PlcToNc <-> Inputs/FromPlc
//   PLC_CRIX_MOT Instance <-> NC-Task 1 SAF/Axes/SL2K2-TOP-M51
//     PlcTask Inputs/Main.M51.Axis.NcToPlc <-> Outputs/ToPlc
//     PlcTask Outputs/Main.M51.Axis.PlcToNc <-> Inputs/FromPlc

// ---- DUTs/Assemblies/ENUM_DiagPaddle.TcDUT
{attribute 'qualified_only'}
{attribute 'strict'}
TYPE ENUM_DiagPaddle :
(
    UNKNOWN := 0,
    PARK :=1,
    UP := 2,
    CENTER := 3,
    PINHOLE := 4,
    DIODE := 5,
    YAG1 := 6,
    YAG2 := 7,
    YAG3 := 8,
    KNIFE := 9
);
END_TYPE

// ---- DUTs/Assemblies/ENUM_DPX.TcDUT
{attribute 'qualified_only'}
// EPICS states enum for use in FB_DPX (diagnostic paddle X)
// Remove strict attribute for easier handling
TYPE ENUM_DPX :
(
    UNKNOWN := 0, // UNKNOWN must be in slot 0 or the FB breaks
    PARK := 1,    // The parked position for the diagnostic paddle
    CENTER := 2,  // center positon for the diagnostic paddle. This should be
    KNIFE	:= 3  // Knife edge position for the diagnostic paddle. Should be the same nominal X positon as the "CENTER"
                  // position, but will use a different set of soft limits to allow scanning of the knife edge.
);
END_TYPE

// ---- DUTs/Assemblies/ENUM_DPY.TcDUT
{attribute 'qualified_only'}
// EPICS states enum for use in FB_DPY (diagnostic paddle Y)
// Remove strict attribute for easier handling
TYPE ENUM_DPY :
(
    UNKNOWN := 0,	// UNKNOWN must be in slot 0 or the FB breaks
    PARK := 1,		// The parked position for the diagnostic paddle
    CENTER := 2,	// center positon for the diagnostic paddle. This should be
    PINHOLE	:= 3,   // Pinhole position for WFS
    DIODE :=4,		// Diode position
    YAG1 := 5,		// Yag 1 position
    YAG2 := 6,		// Yag 2 position
    YAG3 := 7,		// Yag 3 position
    KNIFE := 8 	    // Knife edge position for the diagnostic paddle. Should be the same nominal X positon as the "CENTER"
                    // position, but will use a different set of soft limits to allow scanning of the knife edge.
);
END_TYPE

// ---- DUTs/Assemblies/ENUM_DPZ.TcDUT
{attribute 'qualified_only'}
// EPICS states enum for use in FB_DPX (diagnostic paddle X)
// Remove strict attribute for easier handling
TYPE ENUM_DPZ :
(
    UNKNOWN := 0, // UNKNOWN must be in slot 0 or the FB breaks
    PARK := 1,    // The parked position for the diagnostic paddle
    CENTER := 2  // center positon for the diagnostic paddle. This should be
);
END_TYPE

// ---- DUTs/Assemblies/E_DPaddle_States.TcDUT
{attribute 'qualified_only'}
{attribute 'strict'}
TYPE E_DPaddle_States :
(
    parked := 0,
    diode,
    L1,
    L2,
    L3,
    L4,
    R1,
    R2,
    R3,
    R4
);
END_TYPE

// ---- DUTs/Assemblies/ST_DiagPaddleOutputs.TcDUT
TYPE ST_DiagPaddleOutputs :
STRUCT
    PARK : ARRAY [1..3] OF DUT_PositionState;
    UP : ARRAY [1..3] OF DUT_PositionState;
    CENTER : ARRAY [1..3] OF DUT_PositionState;
    PINHOLE : ARRAY [1..3] OF DUT_PositionState;
    DIODE : ARRAY [1..3] OF DUT_PositionState;
    YAG1 : ARRAY [1..3] OF DUT_PositionState;
    YAG2 : ARRAY [1..3] OF DUT_PositionState;
    YAG3 : ARRAY [1..3] OF DUT_PositionState;
    KNIFE : ARRAY [1..3] OF DUT_PositionState;
END_STRUCT
END_TYPE

// ---- DUTs/EPS/ST_BFSAssemblyState.TcDUT
TYPE ST_BFSAssemblyState :
STRUCT
    iState : DINT;		// state index
    bDiscovered : BOOL;	// BFS search discovery status
    iParent		: DINT;	// BFS parent state

END_STRUCT
END_TYPE

// ---- DUTs/EPS/ST_Queue.TcDUT
TYPE ST_Queue :
STRUCT
    iLength : DINT := 100; // max number of elements in the queue
    iFront	: DINT := 0; // oldest item index
    iBack	: DINT := -1; // newest item index
    iCount	: DINT := 0; // current item count
    arrQueue: ARRAY[0..100] OF ST_BFSAssemblyState; // array to hold queued items
END_STRUCT
END_TYPE

// ---- GVLs/GVL.TcGVL
{attribute 'qualified_only'}
VAR_GLOBAL
    xOverride		:	BOOL := FALSE; // Global override of motion safety settings.
END_VAR

// ---- GVLs/GVL_DiagnosticPaddle.TcGVL
VAR_GLOBAL



    // Define axis states for each axis. These are fed to a FB_PositionState manager for each axis
    // X axis position states
    stDPXPosPark : DUT_PositionState :=		(sName:= 'PARK',
                                             fPosition := 5.0,
                                             fDelta:=1.0,
                                             fVelocity:=5.0,
                                             fAccel:=1.0,
                                            fDecel:=1.0,
                                             bMoveOk:=FALSE,
                                             bLocked:=TRUE,
                                             bValid:=TRUE);
    stDPXPosCenter : DUT_PositionState :=	(sName:= 'CENTER',
                                             fPosition := 10.0,
                                             fDelta:=1.0,
                                             fVelocity:=5.0,
                                             fAccel:=1.0,
                                             fDecel:=1.0,
                                            bMoveOk:=FALSE,
                                             bLocked:=TRUE,
                                             bValid:=TRUE);
    stDPXPosKnife : DUT_PositionState :=	(sName:= 'KNIFE',
                                             fPosition := 15.0,
                                             fDelta:=1.0,
                                             fVelocity:=5.0,
                                             fAccel:=1.0,
                                             fDecel:=1.0,
                                            bMoveOk:=FALSE,
                                             bLocked:=TRUE,
                                             bValid:=TRUE);



    // Y axis position states
    stDPYPosPark : DUT_PositionState :=		(sName:= 'PARK',
                                             fPosition := 5.0,
                                             fDelta:=1.0,
                                             fVelocity:=5.0,
                                             fAccel:=1.0,
                                            fDecel:=1.0,
                                             bMoveOk:=FALSE,
                                             bLocked:=TRUE,
                                             bValid:=TRUE);
    stDPYPosCenter : DUT_PositionState :=	(sName:= 'CENTER',
                                             fPosition := 10.0,
                                             fDelta:=1.0,
                                             fVelocity:=5.0,
                                             fAccel:=1.0,
                                             fDecel:=1.0,
                                            bMoveOk:=FALSE,
                                             bLocked:=TRUE,
                                             bValid:=TRUE);
    stDPYPosDiode : DUT_PositionState :=	(sName:= 'DIODE',
                                             fPosition := 15.0,
                                             fDelta:=1.0,
                                             fVelocity:=5.0,
                                             fAccel:=1.0,
                                            fDecel:=1.0,
                                             bMoveOk:=FALSE,
                                             bLocked:=TRUE,
                                             bValid:=TRUE);
    stDPYPosPinhole : DUT_PositionState :=	(sName:= 'PINHOLE',
                                             fPosition := 20.0,
                                             fDelta:=1.0,
                                             fVelocity:=5.0,
                                             fAccel:=1.0,
                                             fDecel:=1.0,
                                            bMoveOk:=FALSE,
                                             bLocked:=TRUE,
                                             bValid:=TRUE);
    stDPYPosYAG1 : DUT_PositionState :=		(sName:= 'YAG1',
                                             fPosition := 25.0,
                                             fDelta:=1.0,
                                             fVelocity:=5.0,
                                             fAccel:=1.0,
                                             fDecel:=1.0,
                                            bMoveOk:=FALSE,
                                             bLocked:=TRUE,
                                             bValid:=TRUE);
    stDPYPosYAG2 : DUT_PositionState :=		(sName:= 'YAG2',
                                             fPosition := 30.0,
                                             fDelta:=1.0,
                                             fVelocity:=5.0,
                                             fAccel:=1.0,
                                             fDecel:=1.0,
                                            bMoveOk:=FALSE,
                                             bLocked:=TRUE,
                                             bValid:=TRUE);
    stDPYPosYAG3 : DUT_PositionState :=		(sName:= 'YAG3',
                                             fPosition := 35.0,
                                             fDelta:=1.0,
                                             fVelocity:=5.0,
                                             fAccel:=1.0,
                                             fDecel:=1.0,
                                            bMoveOk:=FALSE,
                                             bLocked:=TRUE,
                                             bValid:=TRUE);
    stDPYPosKnife : DUT_PositionState :=	(sName:= 'KNIFE',
                                             fPosition := 40.0,
                                             fDelta:=1.0,
                                             fVelocity:=5.0,
                                             fAccel:=1.0,
                                             fDecel:=1.0,
                                            bMoveOk:=FALSE,
                                             bLocked:=TRUE,
                                             bValid:=TRUE);

    // Z axis position states
    stDPZPosPark : DUT_PositionState :=		(sName:= 'PARK',
                                             fPosition := 5.0,
                                             fDelta:=1.0,
                                             fVelocity:=5.0,
                                             fAccel:=1.0,
                                            fDecel:=1.0,
                                             bMoveOk:=FALSE,
                                             bLocked:=TRUE,
                                             bValid:=TRUE);
    stDPZPosCenter : DUT_PositionState :=	(sName:= 'CENTER',
                                             fPosition := 10.0,
                                             fDelta:=1.0,
                                             fVelocity:=5.0,
                                             fAccel:=1.0,
                                             fDecel:=1.0,
                                            bMoveOk:=FALSE,
                                             bLocked:=TRUE,
                                             bValid:=TRUE);

    stDPPark 	: ST_BFSAssemblyState := (iState:=1, bDiscovered:=FALSE, iParent:=0);
    stDPUp	 	: ST_BFSAssemblyState := (iState:=2, bDiscovered:=FALSE, iParent:=0);
    stDPCenter 	: ST_BFSAssemblyState := (iState:=3, bDiscovered:=FALSE, iParent:=0);
    stDPPinhole : ST_BFSAssemblyState := (iState:=4, bDiscovered:=FALSE, iParent:=0);
    stDPDiode 	: ST_BFSAssemblyState := (iState:=5, bDiscovered:=FALSE, iParent:=0);
    stDPYag1 	: ST_BFSAssemblyState := (iState:=6, bDiscovered:=FALSE, iParent:=0);
    stDPYag2 	: ST_BFSAssemblyState := (iState:=7, bDiscovered:=FALSE, iParent:=0);
    stDPYag3 	: ST_BFSAssemblyState := (iState:=8, bDiscovered:=FALSE, iParent:=0);
    stDPKnife 	: ST_BFSAssemblyState := (iState:=9, bDiscovered:=FALSE, iParent:=0);

    arrDPStates : ARRAY [1..9] OF ST_BFSAssemblyState := [stDPPark, stDPUp, stDPCenter, stDPPinhole, stDPDiode,
                                                          stDPYag1, stDPYag2, stDPYag3, stDPKnife];

END_VAR

// ---- GVLs/GVL_FiberLite.TcGVL
//{attribute 'qualified_only'}
VAR_GLOBAL
    //Fiber-Lite Control
    {attribute 'TcLinkTo' := '.iIlluminatorINT := TIID^Device 1 (EtherCAT)^Term 5 (EK1200)^Term 6 (EK1122-0080)^DRL02-EK0 (EK1101-0080)^DRL02-ECJ1 (EK1122)^CryoStat (EK1101)^Term 158 (EL4004)^AO Outputs Channel 1^Analog output'}
    {attribute 'pytmc' := '
        pv: RIX:CRIX:LED:01
        io: io
    '}
    bLedOutput1 : FB_LED;
END_VAR

// ---- GVLs/GVL_Illumination.TcGVL
//{attribute 'qualified_only'}
VAR_GLOBAL





    // Define axis states for each axis. These are fed to a FB_PositionState manager for each axis
    // X axis position states
    stILMXPosPark : DUT_PositionState :=   (sName:= 'PARK',
                                             fPosition := 0.0,
                                             fDelta:=1.0,
                                             fVelocity:=5.0,
                                             fAccel:=1.0,
                                            fDecel:=1.0,
                                             bMoveOk:=FALSE,
                                             bLocked:=TRUE,
                                             bValid:=TRUE);

    // Y axis position states
    stILMYPosPark : DUT_PositionState :=   (sName:= 'PARK',
                                             fPosition := 0.0,
                                             fDelta:=1.0,
                                             fVelocity:=5.0,
                                             fAccel:=1.0,
                                            fDecel:=1.0,
                                             bMoveOk:=FALSE,
                                             bLocked:=TRUE,
                                             bValid:=TRUE);

    // Z axis position states
    stILMZPosPark : DUT_PositionState :=   (sName:= 'PARK',
                                             fPosition := 0.0,
                                             fDelta:=1.0,
                                             fVelocity:=5.0,
                                             fAccel:=1.0,
                                            fDecel:=1.0,
                                             bMoveOk:=FALSE,
                                             bLocked:=TRUE,
                                             bValid:=TRUE);

    fbILMXStage : FB_MotionStage;
    fbILMYStage : FB_MotionStage;
    fbILMZStage : FB_MotionStage;


END_VAR

// ---- GVLs/GVL_PMPS.TcGVL
{attribute 'qualified_only'}
VAR_GLOBAL
    //MPS
    {attribute 'pytmc' := '
    pv: PLC:CRIX:MOT:FFO:01
    '}
    {attribute 'TcLinkTo' := '.q_xFastFaultOut:=TIIB[PMPS_FFO]^Channel 1^Output'}
    g_FastFaultOutput1  :   FB_HardwareFFOutput :=(i_sNetID:='172.21.42.126.1.1');

    {attribute 'pytmc' := '
    pv: PLC:CRIX:MOT:FFO:02
    '}
    {attribute 'TcLinkTo' := '.q_xFastFaultOut:=TIIB[PMPS_FFO]^Channel 2^Output'}
    g_FastFaultOutput2  :   FB_HardwareFFOutput :=(i_sNetID:='172.21.42.126.1.1');


        {attribute 'pytmc' := '
    pv: PLC:CRIX:MOT:ARB:01
    '}
    fbArbiter1   :   FB_Arbiter(1);
END_VAR

// ---- GVLs/GVL_PointDetector.TcGVL
{attribute 'qualified_only'}
VAR_GLOBAL
        // Motor axes


    // Define axis states for each axis. These are fed to a FB_PositionState manager for each axis
    // Rotation axis position states
    stPDRotPosPark : DUT_PositionState :=		(sName:= 'PARK',
                                             fPosition := 10.0,
                                             fDelta:=1.0,
                                             fVelocity:=5.0,
                                             fAccel:=1.0,
                                            fDecel:=1.0,
                                             bMoveOk:=FALSE,
                                             bLocked:=TRUE,
                                             bValid:=TRUE);

    // Y axis position states
    stPDYPosPark : DUT_PositionState :=		(sName:= 'PARK',
                                             fPosition := 21.0,
                                             fDelta:=1.0,
                                             fVelocity:=5.0,
                                             fAccel:=1.0,
                                            fDecel:=1.0,
                                             bMoveOk:=FALSE,
                                             bLocked:=TRUE,
                                             bValid:=TRUE);

END_VAR

// ---- GVLs/GVL_Questar.TcGVL
{attribute 'qualified_only'}
VAR_GLOBAL
        // Motor axes


    // Define axis states for each axis. These are fed to a FB_PositionState manager for each axis
    // X axis position states
    stQSTXPosPark : DUT_PositionState :=		(sName:= 'PARK',
                                             fPosition := 0.0,
                                             fDelta:=1.0,
                                             fVelocity:=5.0,
                                             fAccel:=1.0,
                                            fDecel:=1.0,
                                             bMoveOk:=FALSE,
                                             bLocked:=TRUE,
                                             bValid:=TRUE);

    // Y axis position states
    stQSTYPosPark : DUT_PositionState :=		(sName:= 'PARK',
                                             fPosition := 0.0,
                                             fDelta:=1.0,
                                             fVelocity:=5.0,
                                             fAccel:=1.0,
                                            fDecel:=1.0,
                                             bMoveOk:=FALSE,
                                             bLocked:=TRUE,
                                             bValid:=TRUE);

END_VAR

// ---- GVLs/GVL_SampleDelivery.TcGVL
{attribute 'qualified_only'}
VAR_GLOBAL
        // Motor axes


    // Define axis states for each axis. These are fed to a FB_PositionState manager for each axis
    // X axis position states
    stSDSXPosPark : DUT_PositionState :=		(sName:= 'PARK',
                                             fPosition := 5.0,
                                             fDelta:=1.0,
                                             fVelocity:=5.0,
                                             fAccel:=1.0,
                                            fDecel:=1.0,
                                             bMoveOk:=FALSE,
                                             bLocked:=TRUE,
                                             bValid:=TRUE);

    // Y axis position states
    stSDSYPosPark : DUT_PositionState :=		(sName:= 'PARK',
                                             fPosition := 5.0,
                                             fDelta:=1.0,
                                             fVelocity:=5.0,
                                             fAccel:=1.0,
                                            fDecel:=1.0,
                                             bMoveOk:=FALSE,
                                             bLocked:=TRUE,
                                             bValid:=TRUE);

    // Z axis position states
    stSDSZPosPark : DUT_PositionState :=		(sName:= 'PARK',
                                             fPosition := 5.0,
                                             fDelta:=1.0,
                                             fVelocity:=5.0,
                                             fAccel:=1.0,
                                            fDecel:=1.0,
                                             bMoveOk:=FALSE,
                                             bLocked:=TRUE,
                                             bValid:=TRUE);
    // Rotation axis position states
    stSDSRotPosPark : DUT_PositionState :=		(sName:= 'PARK',
                                                  fPosition := 5.0,
                                             fDelta:=1.0,
                                             fVelocity:=5.0,
                                             fAccel:=1.0,
                                            fDecel:=1.0,
                                             bMoveOk:=FALSE,
                                             bLocked:=TRUE,
                                             bValid:=TRUE);
    // Shroud axis position states
    stSDSShroudPosPark : DUT_PositionState :=		(sName:= 'PARK',
                                                     fPosition := 5.0,
                                             fDelta:=1.0,
                                             fVelocity:=5.0,
                                             fAccel:=1.0,
                                            fDecel:=1.0,
                                             bMoveOk:=FALSE,
                                             bLocked:=TRUE,
                                             bValid:=TRUE);
END_VAR

// ---- GVLs/Main.TcGVL
	//{attribute 'qualified_only'}
VAR_GLOBAL

    // Motor axes
    {attribute 'pytmc' := 'pv: CRIX:DPL:MMS:X'}
    {attribute 'TcLinkTo' := '.bLimitForwardEnable  := TIID^Device 1 (EtherCAT)^Term 5 (EK1200)^Term 6 (EK1122-0080)^DRL02-EK0 (EK1101-0080)^DRL02-E1 (EL7031)^STM Status^Status^Digital input 2;
                              .bLimitBackwardEnable := TIID^Device 1 (EtherCAT)^Term 5 (EK1200)^Term 6 (EK1122-0080)^DRL02-EK0 (EK1101-0080)^DRL02-E1 (EL7031)^STM Status^Status^Digital input 1'}
    M1 : DUT_MotionStage := (bPowerSelf:=TRUE, nEnableMode:=ENUM_StageEnableMode.DURING_MOTION);
    //stDPXMotor : DUT_MotionStage;

    {attribute 'pytmc' := 'pv: CRIX:DPL:MMS:Y'}
    {attribute 'TcLinkTo' := '.bLimitForwardEnable  := TIID^Device 1 (EtherCAT)^Term 5 (EK1200)^Term 6 (EK1122-0080)^DRL02-EK0 (EK1101-0080)^DRL02-E3 (EL7031)^STM Status^Status^Digital input 1;
                              .bLimitBackwardEnable := TIID^Device 1 (EtherCAT)^Term 5 (EK1200)^Term 6 (EK1122-0080)^DRL02-EK0 (EK1101-0080)^DRL02-E3 (EL7031)^STM Status^Status^Digital input 2'}
    M2 : DUT_MotionStage := (bPowerSelf:=TRUE, nEnableMode:=ENUM_StageEnableMode.DURING_MOTION);
    //stDPYMotor : DUT_MotionStage;

    {attribute 'pytmc' := 'pv: CRIX:DPL:MMS:Z'}
    {attribute 'TcLinkTo' := '.bLimitForwardEnable  := TIID^Device 1 (EtherCAT)^Term 5 (EK1200)^Term 6 (EK1122-0080)^DRL02-EK0 (EK1101-0080)^DRL02-E4 (EL7031)^STM Status^Status^Digital input 1;
                              .bLimitBackwardEnable := TIID^Device 1 (EtherCAT)^Term 5 (EK1200)^Term 6 (EK1122-0080)^DRL02-EK0 (EK1101-0080)^DRL02-E4 (EL7031)^STM Status^Status^Digital input 2'}
    M3 : DUT_MotionStage :=(bPowerSelf:=TRUE,nEnableMode:=ENUM_StageEnableMode.DURING_MOTION);
    //stDPZMotor : DUT_MotionStage;




    {attribute 'pytmc' := 'pv: CRIX:OBJ:MMS:X'}
    {attribute 'TcLinkTo' := '.bLimitForwardEnable  := TIID^Device 1 (EtherCAT)^Term 5 (EK1200)^Term 6 (EK1122-0080)^DRL02-EK0 (EK1101-0080)^DRL02-E6 (EL7031)^STM Status^Status^Digital input 2;
                              .bLimitBackwardEnable := TIID^Device 1 (EtherCAT)^Term 5 (EK1200)^Term 6 (EK1122-0080)^DRL02-EK0 (EK1101-0080)^DRL02-E6 (EL7031)^STM Status^Status^Digital input 1'}
    M4: DUT_MotionStage :=(bPowerSelf:=TRUE ,nEnableMode:=ENUM_StageEnableMode.DURING_MOTION);
    //stOBJXMotor : DUT_MotionStage;

    {attribute 'pytmc' := 'pv: CRIX:OBJ:MMS:Y'}
    {attribute 'TcLinkTo' := '.bLimitForwardEnable  := TIID^Device 1 (EtherCAT)^Term 5 (EK1200)^Term 6 (EK1122-0080)^DRL02-EK0 (EK1101-0080)^DRL02-E7 (EL7031)^STM Status^Status^Digital input 1;
                              .bLimitBackwardEnable := TIID^Device 1 (EtherCAT)^Term 5 (EK1200)^Term 6 (EK1122-0080)^DRL02-EK0 (EK1101-0080)^DRL02-E7 (EL7031)^STM Status^Status^Digital input 2'}
    M5 : DUT_MotionStage :=(bPowerSelf:=TRUE, nEnableMode:=ENUM_StageEnableMode.DURING_MOTION);
    //stOBJYMotor : DUT_MotionStage;

    {attribute 'pytmc' := 'pv: CRIX:OBJ:MMS:Z'}
    {attribute 'TcLinkTo' := '.bLimitForwardEnable  := TIID^Device 1 (EtherCAT)^Term 5 (EK1200)^Term 6 (EK1122-0080)^DRL02-EK0 (EK1101-0080)^DRL02-E9 (EL7031)^STM Status^Status^Digital input 1;
                              .bLimitBackwardEnable := TIID^Device 1 (EtherCAT)^Term 5 (EK1200)^Term 6 (EK1122-0080)^DRL02-EK0 (EK1101-0080)^DRL02-E9 (EL7031)^STM Status^Status^Digital input 2'}
    M6 : DUT_MotionStage :=(bPowerSelf:=TRUE, nEnableMode:=ENUM_StageEnableMode.DURING_MOTION);
    //stOBJZMotor : DUT_MotionStage;



    {attribute 'pytmc' := 'pv: CRIX:PDET:MMS:Y'}
    {attribute 'TcLinkTo' := '.bLimitForwardEnable  := TIID^Device 1 (EtherCAT)^Term 5 (EK1200)^Term 6 (EK1122-0080)^DRL02-EK0 (EK1101-0080)^DRL02-E11 (EL7031)^STM Status^Status^Digital input 1;
                              .bLimitBackwardEnable := TIID^Device 1 (EtherCAT)^Term 5 (EK1200)^Term 6 (EK1122-0080)^DRL02-EK0 (EK1101-0080)^DRL02-E11 (EL7031)^STM Status^Status^Digital input 2'}
    M7 : DUT_MotionStage := (bPowerSelf:=TRUE, nEnableMode:=ENUM_StageEnableMode.DURING_MOTION);
    //stPDYMotor : DUT_MotionStage;
    {attribute 'pytmc' := 'pv: CRIX:PDET:MMS:THETA'}
    {attribute 'TcLinkTo' := '.bLimitForwardEnable  := TIID^Device 1 (EtherCAT)^Term 5 (EK1200)^Term 6 (EK1122-0080)^DRL02-EK0 (EK1101-0080)^DRL02-E13 (EL7041)^STM Status^Status^Digital input 1;
                              .bLimitBackwardEnable := TIID^Device 1 (EtherCAT)^Term 5 (EK1200)^Term 6 (EK1122-0080)^DRL02-EK0 (EK1101-0080)^DRL02-E13 (EL7041)^STM Status^Status^Digital input 2'}
    M8 : DUT_MotionStage := (bPowerSelf:=TRUE, nEnableMode:=ENUM_StageEnableMode.DURING_MOTION);
    //stPDRotMotor : DUT_MotionStage;

    {attribute 'pytmc' := 'pv: CRIX:ILM:MMS:X'}
    {attribute 'TcLinkTo' := '.bLimitForwardEnable  := TIID^Device 1 (EtherCAT)^Term 5 (EK1200)^Term 6 (EK1122-0080)^DRL02-EK0 (EK1101-0080)^Term 65 (EL1084)^Channel 1^Input;
                              .bLimitBackwardEnable := TIID^Device 1 (EtherCAT)^Term 5 (EK1200)^Term 6 (EK1122-0080)^DRL02-EK0 (EK1101-0080)^Term 65 (EL1084)^Channel 2^Input'}
    M9 : DUT_MotionStage := (bPowerSelf:=TRUE, nEnableMode:=ENUM_StageEnableMode.DURING_MOTION); //stILMXMotor : DUT_MotionStage;

    {attribute 'pytmc' := 'pv: CRIX:ILM:MMS:Y'}
    {attribute 'TcLinkTo' := '.bLimitForwardEnable  := TIID^Device 1 (EtherCAT)^Term 5 (EK1200)^Term 6 (EK1122-0080)^DRL02-EK0 (EK1101-0080)^Term 65 (EL1084)^Channel 3^Input;
                              .bLimitBackwardEnable := TIID^Device 1 (EtherCAT)^Term 5 (EK1200)^Term 6 (EK1122-0080)^DRL02-EK0 (EK1101-0080)^Term 65 (EL1084)^Channel 4^Input'}
    M10 : DUT_MotionStage := (bPowerSelf:=TRUE, nEnableMode:=ENUM_StageEnableMode.DURING_MOTION); //stILMYMotor : DUT_MotionStage;

